(* POU GENERAL/ERROR/FB_InitErrorList, ST *)
FUNCTION_BLOCK FB_InitErrorList
VAR_INPUT
END_VAR
VAR_IN_OUT
	T_ErrorList:ST_ERROR_LIST;
END_VAR
VAR_OUTPUT
END_VAR
VAR
END_VAR
(* Static Deutsch Error List *)
T_ErrorList.asErrorListDeutsch.T_LanguagList[1]:='Fehler / Error während disable (Ausschalten) der Station';
T_ErrorList.asErrorListDeutsch.T_LanguagList[2]:='Nicht behandelter undefinierter Station Fehler';
T_ErrorList.asErrorListDeutsch.T_LanguagList[3]:='Z Achse-->Negativer HW Endschalter Aktiv';
T_ErrorList.asErrorListDeutsch.T_LanguagList[4]:='Z Achse-->Positiver HW Endschalter Aktiv';
T_ErrorList.asErrorListDeutsch.T_LanguagList[5]:='Z Achse-->Positiver + Negativer HW Endschalter Aktiv';
T_ErrorList.asErrorListDeutsch.T_LanguagList[6]:='AX5000 Parameter konnte nicht erfolgreich geschrieben werden';
T_ErrorList.asErrorListDeutsch.T_LanguagList[7]:='Achsen MasterModul2 konnte den Spindelkopf L Kanal 1 nicht finden';
T_ErrorList.asErrorListDeutsch.T_LanguagList[8]:='Kalibrierung-->ZylWzAuslenkung Sensor fehlerhaft';
T_ErrorList.asErrorListDeutsch.T_LanguagList[9]:='Z Achse muss referenziert sein';
T_ErrorList.asErrorListDeutsch.T_LanguagList[10]:='Achsen MasterModul2 konnte den Spindelkopf M Kanal 2 nicht finden';
T_ErrorList.asErrorListDeutsch.T_LanguagList[11]:='Hubprozesslänge > Z Mech EndPos';
T_ErrorList.asErrorListDeutsch.T_LanguagList[12]:='Ausfunkhub > Z Mech EndPos';
T_ErrorList.asErrorListDeutsch.T_LanguagList[13]:='Werkzeug ist nicht im Werkstück eingefädelt';
T_ErrorList.asErrorListDeutsch.T_LanguagList[14]:='Kühlmitteldruck ständig vorhanden';
T_ErrorList.asErrorListDeutsch.T_LanguagList[15]:='Fehler 15';
T_ErrorList.asErrorListDeutsch.T_LanguagList[16]:='Beim starten der Bearbeitung darf AuslenkSensor nicht ON sein';
T_ErrorList.asErrorListDeutsch.T_LanguagList[17]:='Beim starten der Bearbeitung darf DrehmSensorHC nicht ON sein';
T_ErrorList.asErrorListDeutsch.T_LanguagList[18]:='Z LadePos > Z Mech EndPos';
T_ErrorList.asErrorListDeutsch.T_LanguagList[19]:='Z Bearb StartPos > Z Mech EndPos';
T_ErrorList.asErrorListDeutsch.T_LanguagList[20]:='Z Bearb EndPos > Z Mech EndPos';
T_ErrorList.asErrorListDeutsch.T_LanguagList[21]:='Z WzWechsel Pos > Z Mech EndPos';
T_ErrorList.asErrorListDeutsch.T_LanguagList[22]:='Z LadePos: Stimmt nicht mit anderen Positionen überein';
T_ErrorList.asErrorListDeutsch.T_LanguagList[23]:='Z Bearb StartPos: Stimmt nicht mit anderen Positionen überein';
T_ErrorList.asErrorListDeutsch.T_LanguagList[24]:='Z Bearb EndPos: Stimmt nicht mit anderen Positionen überein';
T_ErrorList.asErrorListDeutsch.T_LanguagList[25]:='Kalibrierung-->ZylWzAuslenkung Zylinder blockiert';
T_ErrorList.asErrorListDeutsch.T_LanguagList[26]:='Kalibrierung-->ZylWzAuslenkung Sensor fehlerhaft';
T_ErrorList.asErrorListDeutsch.T_LanguagList[27]:='Fehler 27';
T_ErrorList.asErrorListDeutsch.T_LanguagList[28]:='Wz Drehmoment Max überschritten';
T_ErrorList.asErrorListDeutsch.T_LanguagList[29]:='Wz Drehmoment Überlast Aktiv';
T_ErrorList.asErrorListDeutsch.T_LanguagList[30]:='Beim Zentrieren muss der ZylWstkEntspannen auf BearbeitPos sein';
T_ErrorList.asErrorListDeutsch.T_LanguagList[31]:='Z Bearb EndPos Berechn. > Z Bearb EndPos Max';
T_ErrorList.asErrorListDeutsch.T_LanguagList[32]:='Z ZentrierPos berechn. > Z Mech EndPos';
T_ErrorList.asErrorListDeutsch.T_LanguagList[33]:='Zentrier EndPos > Z Mech EndPos';
T_ErrorList.asErrorListDeutsch.T_LanguagList[34]:='Z ZentrierPos berechn. > Z Bearb EndPos Max';
T_ErrorList.asErrorListDeutsch.T_LanguagList[35]:='Z WzZylinder Pos > Z Mech EndPos';
T_ErrorList.asErrorListDeutsch.T_LanguagList[36]:='Beim zylindrischer Teil wurde die Max EndPos erreicht';
T_ErrorList.asErrorListDeutsch.T_LanguagList[37]:='Fehler 37';
T_ErrorList.asErrorListDeutsch.T_LanguagList[38]:='Fehler 38';
T_ErrorList.asErrorListDeutsch.T_LanguagList[39]:='Fehler 39';
T_ErrorList.asErrorListDeutsch.T_LanguagList[40]:='Fehler 40';
T_ErrorList.asErrorListDeutsch.T_LanguagList[41]:='Fehler 41';
T_ErrorList.asErrorListDeutsch.T_LanguagList[42]:='Fehler 42';
T_ErrorList.asErrorListDeutsch.T_LanguagList[43]:='Fehler 43';
T_ErrorList.asErrorListDeutsch.T_LanguagList[44]:='Fehler 44';
T_ErrorList.asErrorListDeutsch.T_LanguagList[45]:='Fehler 45';
T_ErrorList.asErrorListDeutsch.T_LanguagList[46]:='Fehler 46';
T_ErrorList.asErrorListDeutsch.T_LanguagList[47]:='Fehler 47';
T_ErrorList.asErrorListDeutsch.T_LanguagList[48]:='WzWechsel muss vorgenommen werden';
T_ErrorList.asErrorListDeutsch.T_LanguagList[49]:='Datei für zu ladendes Profil nicht gefunden';
T_ErrorList.asErrorListDeutsch.T_LanguagList[50]:='Fehler 50';
T_ErrorList.asErrorListDeutsch.T_LanguagList[51]:='Profilname von Datei ist anders als geladenes Profil';
T_ErrorList.asErrorListDeutsch.T_LanguagList[52]:='Syntaxfehler von zu ladendes Profil';
T_ErrorList.asErrorListDeutsch.T_LanguagList[53]:='Fehler 53';
T_ErrorList.asErrorListDeutsch.T_LanguagList[54]:='Profil konnte nicht gespeichert werden da Verzeichnis fehlt';
T_ErrorList.asErrorListDeutsch.T_LanguagList[55]:='Kalibrierung-->ZylWzDrehmHC Sensor fehlerhaft';
T_ErrorList.asErrorListDeutsch.T_LanguagList[56]:='Kalibrierung-->ZylWzAuslenkung+ZylWzDrehmHC Sensor fehlerhaft';
T_ErrorList.asErrorListDeutsch.T_LanguagList[57]:='Kalibrierung-->ZylWzDrehmHC Zylinder blockiert';
T_ErrorList.asErrorListDeutsch.T_LanguagList[58]:='Kalibrierung-->ZylWzAuslenkung+ZylWzDrehmHC Zylinder blockiert';
T_ErrorList.asErrorListDeutsch.T_LanguagList[59]:='Beim starten der Bearbeitung darf DrehmSensorHCÜberlast nicht ON sein';
T_ErrorList.asErrorListDeutsch.T_LanguagList[60]:='Zentrierproz. HC1 eingetroffen';
T_ErrorList.asErrorListDeutsch.T_LanguagList[61]:='Zentrierproz. StartPos erreicht und HC2 immer noch ON';
T_ErrorList.asErrorListDeutsch.T_LanguagList[62]:='Fehler 62';
T_ErrorList.asErrorListDeutsch.T_LanguagList[63]:='Fehler 63';
T_ErrorList.asErrorListDeutsch.T_LanguagList[64]:='Fehler 64';
T_ErrorList.asErrorListDeutsch.T_LanguagList[65]:='Fehler 65';
T_ErrorList.asErrorListDeutsch.T_LanguagList[66]:='Aufgerufene Achsfunktion besteht nicht';
T_ErrorList.asErrorListDeutsch.T_LanguagList[67]:='Achsfunktion nicht ausführbar wenn Stop-Funktion Aktiv';
T_ErrorList.asErrorListDeutsch.T_LanguagList[68]:='Fehler 68';
T_ErrorList.asErrorListDeutsch.T_LanguagList[69]:='Fehler 69';
T_ErrorList.asErrorListDeutsch.T_LanguagList[70]:='Fehler 70';
T_ErrorList.asErrorListDeutsch.T_LanguagList[71]:='Fehler 71';
T_ErrorList.asErrorListDeutsch.T_LanguagList[72]:='Fehler 72';
T_ErrorList.asErrorListDeutsch.T_LanguagList[73]:='Fehler 73';
T_ErrorList.asErrorListDeutsch.T_LanguagList[74]:='Fehler 74';
T_ErrorList.asErrorListDeutsch.T_LanguagList[75]:='(Schleppabstandsüberschreitung)';
T_ErrorList.asErrorListDeutsch.T_LanguagList[76]:='Not Aus Taste Maschine wurde gedrückt';
T_ErrorList.asErrorListDeutsch.T_LanguagList[77]:='Fehler 77';
T_ErrorList.asErrorListDeutsch.T_LanguagList[78]:='Fehler 78';
T_ErrorList.asErrorListDeutsch.T_LanguagList[79]:='Fehler 79';
T_ErrorList.asErrorListDeutsch.T_LanguagList[80]:='Fehler 80';
T_ErrorList.asErrorListDeutsch.T_LanguagList[81]:='Fehler 81';
T_ErrorList.asErrorListDeutsch.T_LanguagList[82]:='Fehler 82';
T_ErrorList.asErrorListDeutsch.T_LanguagList[83]:='Keine Druckluft';
T_ErrorList.asErrorListDeutsch.T_LanguagList[84]:='EtherCAT 1 Klemme Fehlerhaft';
T_ErrorList.asErrorListDeutsch.T_LanguagList[85]:='EtherCAT 2 Klemme Fehlerhaft';
T_ErrorList.asErrorListDeutsch.T_LanguagList[86]:='Maxon EPOS nicht im Operational Mode OP';
T_ErrorList.asErrorListDeutsch.T_LanguagList[87]:='SMC Ventilinsel nicht im Operational Mode OP';
T_ErrorList.asErrorListDeutsch.T_LanguagList[88]:='Achsen MasterModul 1 nicht im Operational Mode OP';
T_ErrorList.asErrorListDeutsch.T_LanguagList[89]:='Achsen MasterModul 2 nicht im Operational Mode OP';
T_ErrorList.asErrorListDeutsch.T_LanguagList[90]:='Spannungsversorgung 24VDC fehlerhaft';
T_ErrorList.asErrorListDeutsch.T_LanguagList[91]:='Fehler 91';
T_ErrorList.asErrorListDeutsch.T_LanguagList[92]:='Fehler 92';
T_ErrorList.asErrorListDeutsch.T_LanguagList[93]:='Fehler 93';
T_ErrorList.asErrorListDeutsch.T_LanguagList[94]:='Fehler 94';
T_ErrorList.asErrorListDeutsch.T_LanguagList[95]:='Fehler 95';
T_ErrorList.asErrorListDeutsch.T_LanguagList[96]:='Fehler 96';
T_ErrorList.asErrorListDeutsch.T_LanguagList[97]:='Fehler 97';
T_ErrorList.asErrorListDeutsch.T_LanguagList[98]:='USB-Stick konnte nicht gefunden werden für Profil lesen/schreiben';
T_ErrorList.asErrorListDeutsch.T_LanguagList[99]:='USB-Stick konnte nicht gefunden werden für Profil löschen';
T_ErrorList.asErrorListDeutsch.T_LanguagList[100]:='Spannungsversorgung wurde ausgeschaltet';
T_ErrorList.asErrorListDeutsch.T_LanguagList[101]:='Syntaxfehler mindestens einer Profildatei beim lesen aller Profile';
T_ErrorList.asErrorListDeutsch.T_LanguagList[102]:='NovRAM Speicher Fehlerhaft';
T_ErrorList.asErrorListDeutsch.T_LanguagList[103]:='Nicht behandelter undefinierter Prozess Fehler';
T_ErrorList.asErrorListDeutsch.T_LanguagList[104]:='USB-Stick konnte nicht gefunden werden';
T_ErrorList.asErrorListDeutsch.T_LanguagList[105]:='Zylinder Funktion nicht implementiert';
T_ErrorList.asErrorListDeutsch.T_LanguagList[106]:='Zylinder Aktiv-->Sensor nicht ON';
T_ErrorList.asErrorListDeutsch.T_LanguagList[107]:='Zylinder Inaktiv-->Sensor nicht ON';
T_ErrorList.asErrorListDeutsch.T_LanguagList[108]:='Nicht behandelter undefinierter Zylinder Fehler';
T_ErrorList.asErrorListDeutsch.T_LanguagList[109]:='Bremse Aktiv von ST1';
T_ErrorList.asErrorListDeutsch.T_LanguagList[110]:='Fehler 110';
T_ErrorList.asErrorListDeutsch.T_LanguagList[111]:='Fehler 111';
T_ErrorList.asErrorListDeutsch.T_LanguagList[112]:='Fehler 112';
T_ErrorList.asErrorListDeutsch.T_LanguagList[113]:='Fehler 113';
T_ErrorList.asErrorListDeutsch.T_LanguagList[114]:='Fehler 114';
T_ErrorList.asErrorListDeutsch.T_LanguagList[115]:='Fehler 115';
T_ErrorList.asErrorListDeutsch.T_LanguagList[116]:='Fehler 116';
T_ErrorList.asErrorListDeutsch.T_LanguagList[117]:='Fehler 117';
T_ErrorList.asErrorListDeutsch.T_LanguagList[118]:='Fehler 118';
T_ErrorList.asErrorListDeutsch.T_LanguagList[119]:='Fehler 119';
T_ErrorList.asErrorListDeutsch.T_LanguagList[120]:='Fehler 120';
T_ErrorList.asErrorListDeutsch.T_LanguagList[121]:='Fehler 121';
T_ErrorList.asErrorListDeutsch.T_LanguagList[122]:='Fehler 122';
T_ErrorList.asErrorListDeutsch.T_LanguagList[123]:='Fehler 123';
T_ErrorList.asErrorListDeutsch.T_LanguagList[124]:='Fehler 124';
T_ErrorList.asErrorListDeutsch.T_LanguagList[125]:='Fehler 125';
T_ErrorList.asErrorListDeutsch.T_LanguagList[126]:='Fehler 126';
T_ErrorList.asErrorListDeutsch.T_LanguagList[127]:='Fehler 127';
T_ErrorList.asErrorListDeutsch.T_LanguagList[128]:='Fehler 128';
T_ErrorList.asErrorListDeutsch.T_LanguagList[129]:='Fehler 129';
T_ErrorList.asErrorListDeutsch.T_LanguagList[130]:='Fehler 130';
T_ErrorList.asErrorListDeutsch.T_LanguagList[131]:='Fehler 131';
T_ErrorList.asErrorListDeutsch.T_LanguagList[132]:='Fehler 132';
T_ErrorList.asErrorListDeutsch.T_LanguagList[133]:='Fehler 133';
T_ErrorList.asErrorListDeutsch.T_LanguagList[134]:='Fehler 134';
T_ErrorList.asErrorListDeutsch.T_LanguagList[135]:='Fehler 135';
T_ErrorList.asErrorListDeutsch.T_LanguagList[136]:='Fehler 136';
T_ErrorList.asErrorListDeutsch.T_LanguagList[137]:='Fehler 137';
T_ErrorList.asErrorListDeutsch.T_LanguagList[138]:='Fehler 138';
T_ErrorList.asErrorListDeutsch.T_LanguagList[139]:='Fehler 139';
T_ErrorList.asErrorListDeutsch.T_LanguagList[140]:='Fehler 140';
T_ErrorList.asErrorListDeutsch.T_LanguagList[141]:='Fehler 141';
T_ErrorList.asErrorListDeutsch.T_LanguagList[142]:='Fehler 142';
T_ErrorList.asErrorListDeutsch.T_LanguagList[143]:='Fehler 143';
T_ErrorList.asErrorListDeutsch.T_LanguagList[144]:='Fehler 144';
T_ErrorList.asErrorListDeutsch.T_LanguagList[145]:='Fehler 145';
T_ErrorList.asErrorListDeutsch.T_LanguagList[146]:='HDD steht nicht Bereit';
T_ErrorList.asErrorListDeutsch.T_LanguagList[147]:='Timeout beim Schreiben auf USB-Stick';
T_ErrorList.asErrorListDeutsch.T_LanguagList[148]:='USB Stick nicht schreibbar';
T_ErrorList.asErrorListDeutsch.T_LanguagList[149]:='USB Stick nicht gefunden';
T_ErrorList.asErrorListDeutsch.T_LanguagList[150]:='Fehler 150';
T_ErrorList.asErrorListDeutsch.T_LanguagList[151]:='Fehler 151';
T_ErrorList.asErrorListDeutsch.T_LanguagList[152]:='Fehler 152';
T_ErrorList.asErrorListDeutsch.T_LanguagList[153]:='Fehler 153';
T_ErrorList.asErrorListDeutsch.T_LanguagList[154]:='Fehler 154';
T_ErrorList.asErrorListDeutsch.T_LanguagList[155]:='Fehler 155';
T_ErrorList.asErrorListDeutsch.T_LanguagList[156]:='Fehler 156';
T_ErrorList.asErrorListDeutsch.T_LanguagList[157]:='Fehler 157';
T_ErrorList.asErrorListDeutsch.T_LanguagList[158]:='Fehler 158';
T_ErrorList.asErrorListDeutsch.T_LanguagList[159]:='Fehler 159';
T_ErrorList.asErrorListDeutsch.T_LanguagList[160]:='Fehler 160';
T_ErrorList.asErrorListDeutsch.T_LanguagList[161]:='Fehler 161';
T_ErrorList.asErrorListDeutsch.T_LanguagList[162]:='Fehler 162';
T_ErrorList.asErrorListDeutsch.T_LanguagList[163]:='Fehler 163';
T_ErrorList.asErrorListDeutsch.T_LanguagList[164]:='Fehler 164';
T_ErrorList.asErrorListDeutsch.T_LanguagList[165]:='Fehler 165';
T_ErrorList.asErrorListDeutsch.T_LanguagList[166]:='Fehler 166';
T_ErrorList.asErrorListDeutsch.T_LanguagList[167]:='Fehler 167';
T_ErrorList.asErrorListDeutsch.T_LanguagList[168]:='Fehler 168';
T_ErrorList.asErrorListDeutsch.T_LanguagList[169]:='Fehler 169';
T_ErrorList.asErrorListDeutsch.T_LanguagList[170]:='Fehler 170';
T_ErrorList.asErrorListDeutsch.T_LanguagList[171]:='Fehler 171';
T_ErrorList.asErrorListDeutsch.T_LanguagList[172]:='Fehler 172';
T_ErrorList.asErrorListDeutsch.T_LanguagList[173]:='Fehler 173';
T_ErrorList.asErrorListDeutsch.T_LanguagList[174]:='Fehler 174';
T_ErrorList.asErrorListDeutsch.T_LanguagList[175]:='Fehler 175';
T_ErrorList.asErrorListDeutsch.T_LanguagList[176]:='Fehler 176';
T_ErrorList.asErrorListDeutsch.T_LanguagList[177]:='Fehler 177';
T_ErrorList.asErrorListDeutsch.T_LanguagList[178]:='Fehler 178';
T_ErrorList.asErrorListDeutsch.T_LanguagList[179]:='Fehler 179';
T_ErrorList.asErrorListDeutsch.T_LanguagList[180]:='Fehler 180';
T_ErrorList.asErrorListDeutsch.T_LanguagList[181]:='Fehler 181';
T_ErrorList.asErrorListDeutsch.T_LanguagList[182]:='Fehler 182';
T_ErrorList.asErrorListDeutsch.T_LanguagList[183]:='Fehler 183';
T_ErrorList.asErrorListDeutsch.T_LanguagList[184]:='Fehler 184';
T_ErrorList.asErrorListDeutsch.T_LanguagList[185]:='Fehler 185';
T_ErrorList.asErrorListDeutsch.T_LanguagList[186]:='Fehler 186';
T_ErrorList.asErrorListDeutsch.T_LanguagList[187]:='Fehler 187';
T_ErrorList.asErrorListDeutsch.T_LanguagList[188]:='Fehler 188';
T_ErrorList.asErrorListDeutsch.T_LanguagList[189]:='Fehler 189';
T_ErrorList.asErrorListDeutsch.T_LanguagList[190]:='Fehler 190';
T_ErrorList.asErrorListDeutsch.T_LanguagList[191]:='Fehler 191';
T_ErrorList.asErrorListDeutsch.T_LanguagList[192]:='Fehler 192';
T_ErrorList.asErrorListDeutsch.T_LanguagList[193]:='Fehler 193';
T_ErrorList.asErrorListDeutsch.T_LanguagList[194]:='Fehler 194';
T_ErrorList.asErrorListDeutsch.T_LanguagList[195]:='Fehler 195';
T_ErrorList.asErrorListDeutsch.T_LanguagList[196]:='Fehler 196';
T_ErrorList.asErrorListDeutsch.T_LanguagList[197]:='Fehler 197';
T_ErrorList.asErrorListDeutsch.T_LanguagList[198]:='Fehler 198';
T_ErrorList.asErrorListDeutsch.T_LanguagList[199]:='Fehler 199';
T_ErrorList.asErrorListDeutsch.T_LanguagList[200]:='Fehler 200';
T_ErrorList.asErrorListDeutsch.T_LanguagList[201]:='Fehler 201';
T_ErrorList.asErrorListDeutsch.T_LanguagList[202]:='Fehler 202';
T_ErrorList.asErrorListDeutsch.T_LanguagList[203]:='Fehler 203';
T_ErrorList.asErrorListDeutsch.T_LanguagList[204]:='Fehler 204';
T_ErrorList.asErrorListDeutsch.T_LanguagList[205]:='Fehler 205';
T_ErrorList.asErrorListDeutsch.T_LanguagList[206]:='Fehler 206';
T_ErrorList.asErrorListDeutsch.T_LanguagList[207]:='Fehler 207';
T_ErrorList.asErrorListDeutsch.T_LanguagList[208]:='Fehler 208';
T_ErrorList.asErrorListDeutsch.T_LanguagList[209]:='Fehler 209';
T_ErrorList.asErrorListDeutsch.T_LanguagList[210]:='Fehler 210';
T_ErrorList.asErrorListDeutsch.T_LanguagList[211]:='Fehler 211';
T_ErrorList.asErrorListDeutsch.T_LanguagList[212]:='Fehler 212';
T_ErrorList.asErrorListDeutsch.T_LanguagList[213]:='Fehler 213';
T_ErrorList.asErrorListDeutsch.T_LanguagList[214]:='Fehler 214';
T_ErrorList.asErrorListDeutsch.T_LanguagList[215]:='Fehler 215';
T_ErrorList.asErrorListDeutsch.T_LanguagList[216]:='Fehler 216';
T_ErrorList.asErrorListDeutsch.T_LanguagList[217]:='Fehler 217';
T_ErrorList.asErrorListDeutsch.T_LanguagList[218]:='Fehler 218';
T_ErrorList.asErrorListDeutsch.T_LanguagList[219]:='Fehler 219';
T_ErrorList.asErrorListDeutsch.T_LanguagList[220]:='Fehler 220';
T_ErrorList.asErrorListDeutsch.T_LanguagList[221]:='Fehler 221';
T_ErrorList.asErrorListDeutsch.T_LanguagList[222]:='Fehler 222';
T_ErrorList.asErrorListDeutsch.T_LanguagList[223]:='Fehler 223';
T_ErrorList.asErrorListDeutsch.T_LanguagList[224]:='Fehler 224';
T_ErrorList.asErrorListDeutsch.T_LanguagList[225]:='Fehler 225';
T_ErrorList.asErrorListDeutsch.T_LanguagList[226]:='Fehler 226';
T_ErrorList.asErrorListDeutsch.T_LanguagList[227]:='Fehler 227';
T_ErrorList.asErrorListDeutsch.T_LanguagList[228]:='Fehler 228';
T_ErrorList.asErrorListDeutsch.T_LanguagList[229]:='Fehler 229';
T_ErrorList.asErrorListDeutsch.T_LanguagList[230]:='Fehler 230';
T_ErrorList.asErrorListDeutsch.T_LanguagList[231]:='Fehler 231';
T_ErrorList.asErrorListDeutsch.T_LanguagList[232]:='Fehler 232';
T_ErrorList.asErrorListDeutsch.T_LanguagList[233]:='Fehler 233';
T_ErrorList.asErrorListDeutsch.T_LanguagList[234]:='Fehler 234';
T_ErrorList.asErrorListDeutsch.T_LanguagList[235]:='Fehler 235';
T_ErrorList.asErrorListDeutsch.T_LanguagList[236]:='Fehler 236';
T_ErrorList.asErrorListDeutsch.T_LanguagList[237]:='Fehler 237';
T_ErrorList.asErrorListDeutsch.T_LanguagList[238]:='Fehler 238';
T_ErrorList.asErrorListDeutsch.T_LanguagList[239]:='Fehler 239';
T_ErrorList.asErrorListDeutsch.T_LanguagList[240]:='Fehler 240';
T_ErrorList.asErrorListDeutsch.T_LanguagList[241]:='Fehler 241';
T_ErrorList.asErrorListDeutsch.T_LanguagList[242]:='Fehler 242';
T_ErrorList.asErrorListDeutsch.T_LanguagList[243]:='Fehler 243';
T_ErrorList.asErrorListDeutsch.T_LanguagList[244]:='Fehler 244';
T_ErrorList.asErrorListDeutsch.T_LanguagList[245]:='Fehler 245';
T_ErrorList.asErrorListDeutsch.T_LanguagList[246]:='Fehler 246';
T_ErrorList.asErrorListDeutsch.T_LanguagList[247]:='Fehler 247';
T_ErrorList.asErrorListDeutsch.T_LanguagList[248]:='Fehler 248';
T_ErrorList.asErrorListDeutsch.T_LanguagList[249]:='Fehler 249';
T_ErrorList.asErrorListDeutsch.T_LanguagList[250]:='Fehler 250';
T_ErrorList.asErrorListDeutsch.T_LanguagList[251]:='Fehler 251';
T_ErrorList.asErrorListDeutsch.T_LanguagList[252]:='Fehler 252';
T_ErrorList.asErrorListDeutsch.T_LanguagList[253]:='Fehler 253';
T_ErrorList.asErrorListDeutsch.T_LanguagList[254]:='Fehler 254';
T_ErrorList.asErrorListDeutsch.T_LanguagList[255]:='Fehler 255';
T_ErrorList.asErrorListDeutsch.T_LanguagList[256]:='Fehler 256';
T_ErrorList.asErrorListDeutsch.T_LanguagList[257]:='Fehler 257';
T_ErrorList.asErrorListDeutsch.T_LanguagList[258]:='Fehler 258';
T_ErrorList.asErrorListDeutsch.T_LanguagList[259]:='Fehler 259';
T_ErrorList.asErrorListDeutsch.T_LanguagList[260]:='Fehler 260';
T_ErrorList.asErrorListDeutsch.T_LanguagList[261]:='Fehler 261';
T_ErrorList.asErrorListDeutsch.T_LanguagList[262]:='Fehler 262';
T_ErrorList.asErrorListDeutsch.T_LanguagList[263]:='Fehler 263';
T_ErrorList.asErrorListDeutsch.T_LanguagList[264]:='Fehler 264';
T_ErrorList.asErrorListDeutsch.T_LanguagList[265]:='Fehler 265';
T_ErrorList.asErrorListDeutsch.T_LanguagList[266]:='Fehler 266';
T_ErrorList.asErrorListDeutsch.T_LanguagList[267]:='Fehler 267';
T_ErrorList.asErrorListDeutsch.T_LanguagList[268]:='Fehler 268';
T_ErrorList.asErrorListDeutsch.T_LanguagList[269]:='Fehler 269';
T_ErrorList.asErrorListDeutsch.T_LanguagList[270]:='Fehler 270';
T_ErrorList.asErrorListDeutsch.T_LanguagList[271]:='Fehler 271';
T_ErrorList.asErrorListDeutsch.T_LanguagList[272]:='Fehler 272';
T_ErrorList.asErrorListDeutsch.T_LanguagList[273]:='Fehler 273';
T_ErrorList.asErrorListDeutsch.T_LanguagList[274]:='Fehler 274';
T_ErrorList.asErrorListDeutsch.T_LanguagList[275]:='Fehler 275';
T_ErrorList.asErrorListDeutsch.T_LanguagList[276]:='Fehler 276';
T_ErrorList.asErrorListDeutsch.T_LanguagList[277]:='Fehler 277';
T_ErrorList.asErrorListDeutsch.T_LanguagList[278]:='Fehler 278';
T_ErrorList.asErrorListDeutsch.T_LanguagList[279]:='Fehler 279';
T_ErrorList.asErrorListDeutsch.T_LanguagList[280]:='Fehler 280';
T_ErrorList.asErrorListDeutsch.T_LanguagList[281]:='Fehler 281';
T_ErrorList.asErrorListDeutsch.T_LanguagList[282]:='Fehler 282';
T_ErrorList.asErrorListDeutsch.T_LanguagList[283]:='Fehler 283';
T_ErrorList.asErrorListDeutsch.T_LanguagList[284]:='Fehler 284';
T_ErrorList.asErrorListDeutsch.T_LanguagList[285]:='Fehler 285';
T_ErrorList.asErrorListDeutsch.T_LanguagList[286]:='Fehler 286';
T_ErrorList.asErrorListDeutsch.T_LanguagList[287]:='Fehler 287';
T_ErrorList.asErrorListDeutsch.T_LanguagList[288]:='Fehler 288';
T_ErrorList.asErrorListDeutsch.T_LanguagList[289]:='Fehler 289';
T_ErrorList.asErrorListDeutsch.T_LanguagList[290]:='Fehler 290';
T_ErrorList.asErrorListDeutsch.T_LanguagList[291]:='Fehler 291';
T_ErrorList.asErrorListDeutsch.T_LanguagList[292]:='Fehler 292';
T_ErrorList.asErrorListDeutsch.T_LanguagList[293]:='Fehler 293';
T_ErrorList.asErrorListDeutsch.T_LanguagList[294]:='Fehler 294';
T_ErrorList.asErrorListDeutsch.T_LanguagList[295]:='Fehler 295';
T_ErrorList.asErrorListDeutsch.T_LanguagList[296]:='Fehler 296';
T_ErrorList.asErrorListDeutsch.T_LanguagList[297]:='Fehler 297';
T_ErrorList.asErrorListDeutsch.T_LanguagList[298]:='Fehler 298';
T_ErrorList.asErrorListDeutsch.T_LanguagList[299]:='Fehler 299';
T_ErrorList.asErrorListDeutsch.T_LanguagList[300]:='Fehler 300';

(* Static English Error List *)
T_ErrorList.asErrorListEnglish.T_LanguagList[1]:='Error while disable of the Station';
T_ErrorList.asErrorListEnglish.T_LanguagList[2]:='Not handled undefined Station Error';
T_ErrorList.asErrorListEnglish.T_LanguagList[3]:='Z Axis-->Negative HW limit switch Active';
T_ErrorList.asErrorListEnglish.T_LanguagList[4]:='Z Axis-->Positive HW limit switch Active';
T_ErrorList.asErrorListEnglish.T_LanguagList[5]:='Z Axis-->Positive + Negative HW limit switch Active';
T_ErrorList.asErrorListEnglish.T_LanguagList[6]:='AX5000 Parameter could not be written successfully';
T_ErrorList.asErrorListEnglish.T_LanguagList[7]:='Axis MasterModul2 could not find spindle head L channel 1';
T_ErrorList.asErrorListEnglish.T_LanguagList[8]:='Calibration-->CylToolDeflection Sensor failure';
T_ErrorList.asErrorListEnglish.T_LanguagList[9]:='Z Axis must be referenced';
T_ErrorList.asErrorListEnglish.T_LanguagList[10]:='Axis MasterModul2 could not find spindle head M channel 2';
T_ErrorList.asErrorListEnglish.T_LanguagList[11]:='Z Process stroke > Z Mech EndPos';
T_ErrorList.asErrorListEnglish.T_LanguagList[12]:='Spark-out > Z Mech EndPos';
T_ErrorList.asErrorListEnglish.T_LanguagList[13]:='Tool is not Infeeded into the Workpiece';
T_ErrorList.asErrorListEnglish.T_LanguagList[14]:='Coolant pressure still ON';
T_ErrorList.asErrorListEnglish.T_LanguagList[15]:='Error 15';
T_ErrorList.asErrorListEnglish.T_LanguagList[16]:='During starting of the Working could not be ON the ToolDeflection Sensor';
T_ErrorList.asErrorListEnglish.T_LanguagList[17]:='During starting of the Working could not be ON the ToolTorque Sensor';
T_ErrorList.asErrorListEnglish.T_LanguagList[18]:='Z LoadPos > Z Mech EndPos';
T_ErrorList.asErrorListEnglish.T_LanguagList[19]:='Z Work StartPos > Z Mech EndPos';
T_ErrorList.asErrorListEnglish.T_LanguagList[20]:='Z Work EndPos > Z Mech EndPos';
T_ErrorList.asErrorListEnglish.T_LanguagList[21]:='Z ToolChange Pos > Z Mech EndPos';
T_ErrorList.asErrorListEnglish.T_LanguagList[22]:='Z LoadPos: Discrepancy with other Z Position';
T_ErrorList.asErrorListEnglish.T_LanguagList[23]:='Z Work StartPos: Discrepancy with other Z Position';
T_ErrorList.asErrorListEnglish.T_LanguagList[24]:='Z Work EndPos: Discrepancy with other Z Position';
T_ErrorList.asErrorListEnglish.T_LanguagList[25]:='Calibration-->CylToolDeflection Cylinder is blocked';
T_ErrorList.asErrorListEnglish.T_LanguagList[26]:='Calibration-->CylToolDeflection Sensor failure';
T_ErrorList.asErrorListEnglish.T_LanguagList[27]:='Error 27';
T_ErrorList.asErrorListEnglish.T_LanguagList[28]:='ToolTorque Max exceed';
T_ErrorList.asErrorListEnglish.T_LanguagList[29]:='ToolTorque Overload Active';
T_ErrorList.asErrorListEnglish.T_LanguagList[30]:='When centring, the CylWPUnfix must be to WorkPosition';
T_ErrorList.asErrorListEnglish.T_LanguagList[31]:='Z Work EndPos calc. > Z Work EndPos Max';
T_ErrorList.asErrorListEnglish.T_LanguagList[32]:='Z Centring Pos calc. > Z Mech EndPos';
T_ErrorList.asErrorListEnglish.T_LanguagList[33]:='Z Centring EndPos > Z Mech EndPos';
T_ErrorList.asErrorListEnglish.T_LanguagList[34]:='Z Centring Pos calc. > Z Work EndPos Max';
T_ErrorList.asErrorListEnglish.T_LanguagList[35]:='Z ToolCylindrical Pos > Z Mech EndPos';
T_ErrorList.asErrorListEnglish.T_LanguagList[36]:='On cylindrical part was reach the max EndPos';
T_ErrorList.asErrorListEnglish.T_LanguagList[37]:='Error 37';
T_ErrorList.asErrorListEnglish.T_LanguagList[38]:='Error 38';
T_ErrorList.asErrorListEnglish.T_LanguagList[39]:='Error 39';
T_ErrorList.asErrorListEnglish.T_LanguagList[40]:='Error 40';
T_ErrorList.asErrorListEnglish.T_LanguagList[41]:='Error 41';
T_ErrorList.asErrorListEnglish.T_LanguagList[42]:='Error 42';
T_ErrorList.asErrorListEnglish.T_LanguagList[43]:='Error 43';
T_ErrorList.asErrorListEnglish.T_LanguagList[44]:='Error 44';
T_ErrorList.asErrorListEnglish.T_LanguagList[45]:='Error 45';
T_ErrorList.asErrorListEnglish.T_LanguagList[46]:='Error 46';
T_ErrorList.asErrorListEnglish.T_LanguagList[47]:='Error 47';
T_ErrorList.asErrorListEnglish.T_LanguagList[48]:='Tool must be changed';
T_ErrorList.asErrorListEnglish.T_LanguagList[49]:='File for to load Profile not found';
T_ErrorList.asErrorListEnglish.T_LanguagList[50]:='Error 50';
T_ErrorList.asErrorListEnglish.T_LanguagList[51]:='Profile name of File is different as loaded Profile';
T_ErrorList.asErrorListEnglish.T_LanguagList[52]:='Syntax Error of to load Profile';
T_ErrorList.asErrorListEnglish.T_LanguagList[53]:='Error 53';
T_ErrorList.asErrorListEnglish.T_LanguagList[54]:='Profile not saved because the directory is missing';
T_ErrorList.asErrorListEnglish.T_LanguagList[55]:='Calibration-->CylToolTorque Sensor failure';
T_ErrorList.asErrorListEnglish.T_LanguagList[56]:='Calibration-->CylToolDeflection+CylToolTorque Sensor failure';
T_ErrorList.asErrorListEnglish.T_LanguagList[57]:='Calibration-->CylToolTorque Cylinder is blocked';
T_ErrorList.asErrorListEnglish.T_LanguagList[58]:='Calibration-->CylToolDeflection+CylToolTorque Cylinder is blocked';
T_ErrorList.asErrorListEnglish.T_LanguagList[59]:='During starting of the Working could not be ON the ToolTorque Overload Sensor';
T_ErrorList.asErrorListEnglish.T_LanguagList[60]:='Centring Process HC1 active';
T_ErrorList.asErrorListEnglish.T_LanguagList[61]:='Centring Proc. StartPos reach and HC2 still ON';
T_ErrorList.asErrorListEnglish.T_LanguagList[62]:='Error 62';
T_ErrorList.asErrorListEnglish.T_LanguagList[63]:='Error 63';
T_ErrorList.asErrorListEnglish.T_LanguagList[64]:='Error 64';
T_ErrorList.asErrorListEnglish.T_LanguagList[65]:='Error 65';
T_ErrorList.asErrorListEnglish.T_LanguagList[66]:='Called Axis function do not exist';
T_ErrorList.asErrorListEnglish.T_LanguagList[67]:='Axis function not executable during Stopp- function is Active';
T_ErrorList.asErrorListEnglish.T_LanguagList[68]:='Error 68';
T_ErrorList.asErrorListEnglish.T_LanguagList[69]:='Error 69';
T_ErrorList.asErrorListEnglish.T_LanguagList[70]:='Error 70';
T_ErrorList.asErrorListEnglish.T_LanguagList[71]:='Error 71';
T_ErrorList.asErrorListEnglish.T_LanguagList[72]:='Error 72';
T_ErrorList.asErrorListEnglish.T_LanguagList[73]:='Error 73';
T_ErrorList.asErrorListEnglish.T_LanguagList[74]:='Error 74';
T_ErrorList.asErrorListEnglish.T_LanguagList[75]:='(Position drag excess)';
T_ErrorList.asErrorListEnglish.T_LanguagList[76]:='Emergency Button Machine pressed';
T_ErrorList.asErrorListEnglish.T_LanguagList[77]:='Error 77';
T_ErrorList.asErrorListEnglish.T_LanguagList[78]:='Error 78';
T_ErrorList.asErrorListEnglish.T_LanguagList[79]:='Error 79';
T_ErrorList.asErrorListEnglish.T_LanguagList[80]:='Error 80';
T_ErrorList.asErrorListEnglish.T_LanguagList[81]:='Error 81';
T_ErrorList.asErrorListEnglish.T_LanguagList[82]:='Error 82';
T_ErrorList.asErrorListEnglish.T_LanguagList[83]:='No air pressure';
T_ErrorList.asErrorListEnglish.T_LanguagList[84]:='EtherCAT 1 Terminal failure';
T_ErrorList.asErrorListEnglish.T_LanguagList[85]:='EtherCAT 2 Terminal failure';
T_ErrorList.asErrorListEnglish.T_LanguagList[86]:='Maxon EPOS not in Operational Mode OP';
T_ErrorList.asErrorListEnglish.T_LanguagList[87]:='SMC Valve not in Operational Mode OP';
T_ErrorList.asErrorListEnglish.T_LanguagList[88]:='Axis MasterModul 1 not in Operational Mode OP';
T_ErrorList.asErrorListEnglish.T_LanguagList[89]:='Axis MasterModul 2 not in Operational Mode OP';
T_ErrorList.asErrorListEnglish.T_LanguagList[90]:='Power 24VDC failure';
T_ErrorList.asErrorListEnglish.T_LanguagList[91]:='Error 91';
T_ErrorList.asErrorListEnglish.T_LanguagList[92]:='Error 92';
T_ErrorList.asErrorListEnglish.T_LanguagList[93]:='Error 93';
T_ErrorList.asErrorListEnglish.T_LanguagList[94]:='Error 94';
T_ErrorList.asErrorListEnglish.T_LanguagList[95]:='Error 95';
T_ErrorList.asErrorListEnglish.T_LanguagList[96]:='Error 96';
T_ErrorList.asErrorListEnglish.T_LanguagList[97]:='Error 97';
T_ErrorList.asErrorListEnglish.T_LanguagList[98]:='USB-Stick not founded for Profile read/write';
T_ErrorList.asErrorListEnglish.T_LanguagList[99]:='USB-Stick not founded for Profile delete';
T_ErrorList.asErrorListEnglish.T_LanguagList[100]:='Power Supply is switched off';
T_ErrorList.asErrorListEnglish.T_LanguagList[101]:='At least one Profle has a syntax Error during reading of all Profiles';
T_ErrorList.asErrorListEnglish.T_LanguagList[102]:='NovRAM store failure';
T_ErrorList.asErrorListEnglish.T_LanguagList[103]:='Not handled undefined Process Error';
T_ErrorList.asErrorListEnglish.T_LanguagList[104]:='USB-Stick not founded';
T_ErrorList.asErrorListEnglish.T_LanguagList[105]:='Cylinder function not implemented';
T_ErrorList.asErrorListEnglish.T_LanguagList[106]:='Cylinder Active-->Sensor not ON';
T_ErrorList.asErrorListEnglish.T_LanguagList[107]:='Cylinder Inactive-->Sensor not ON';
T_ErrorList.asErrorListEnglish.T_LanguagList[108]:='Not handled undefined Cylinder Error';
T_ErrorList.asErrorListEnglish.T_LanguagList[109]:='Axis Brake Active of ST1';
T_ErrorList.asErrorListEnglish.T_LanguagList[110]:='Error 110';
T_ErrorList.asErrorListEnglish.T_LanguagList[111]:='Error 111';
T_ErrorList.asErrorListEnglish.T_LanguagList[112]:='Error 112';
T_ErrorList.asErrorListEnglish.T_LanguagList[113]:='Error 113';
T_ErrorList.asErrorListEnglish.T_LanguagList[114]:='Error 114';
T_ErrorList.asErrorListEnglish.T_LanguagList[115]:='Error 115';
T_ErrorList.asErrorListEnglish.T_LanguagList[116]:='Error 116';
T_ErrorList.asErrorListEnglish.T_LanguagList[117]:='Error 117';
T_ErrorList.asErrorListEnglish.T_LanguagList[118]:='Error 118';
T_ErrorList.asErrorListEnglish.T_LanguagList[119]:='Error 119';
T_ErrorList.asErrorListEnglish.T_LanguagList[120]:='Error 120';
T_ErrorList.asErrorListEnglish.T_LanguagList[121]:='Error 121';
T_ErrorList.asErrorListEnglish.T_LanguagList[122]:='Error 122';
T_ErrorList.asErrorListEnglish.T_LanguagList[123]:='Error 123';
T_ErrorList.asErrorListEnglish.T_LanguagList[124]:='Error 124';
T_ErrorList.asErrorListEnglish.T_LanguagList[125]:='Error 125';
T_ErrorList.asErrorListEnglish.T_LanguagList[126]:='Error 126';
T_ErrorList.asErrorListEnglish.T_LanguagList[127]:='Error 127';
T_ErrorList.asErrorListEnglish.T_LanguagList[128]:='Error 128';
T_ErrorList.asErrorListEnglish.T_LanguagList[129]:='Error 129';
T_ErrorList.asErrorListEnglish.T_LanguagList[130]:='Error 130';
T_ErrorList.asErrorListEnglish.T_LanguagList[131]:='Error 131';
T_ErrorList.asErrorListEnglish.T_LanguagList[132]:='Error 132';
T_ErrorList.asErrorListEnglish.T_LanguagList[133]:='Error 133';
T_ErrorList.asErrorListEnglish.T_LanguagList[134]:='Error 134';
T_ErrorList.asErrorListEnglish.T_LanguagList[135]:='Error 135';
T_ErrorList.asErrorListEnglish.T_LanguagList[136]:='Error 136';
T_ErrorList.asErrorListEnglish.T_LanguagList[137]:='Error 137';
T_ErrorList.asErrorListEnglish.T_LanguagList[138]:='Error 138';
T_ErrorList.asErrorListEnglish.T_LanguagList[139]:='Error 139';
T_ErrorList.asErrorListEnglish.T_LanguagList[140]:='Error 140';
T_ErrorList.asErrorListEnglish.T_LanguagList[141]:='Error 141';
T_ErrorList.asErrorListEnglish.T_LanguagList[142]:='Error 142';
T_ErrorList.asErrorListEnglish.T_LanguagList[143]:='Error 143';
T_ErrorList.asErrorListEnglish.T_LanguagList[144]:='Error 144';
T_ErrorList.asErrorListEnglish.T_LanguagList[145]:='Error 145';
T_ErrorList.asErrorListEnglish.T_LanguagList[146]:='HDD not Ready';
T_ErrorList.asErrorListEnglish.T_LanguagList[147]:='Timeout while write on USB-Stick';
T_ErrorList.asErrorListEnglish.T_LanguagList[148]:='USB Stick no writing';
T_ErrorList.asErrorListEnglish.T_LanguagList[149]:='USB Stick not found';
T_ErrorList.asErrorListEnglish.T_LanguagList[150]:='Error 150';
T_ErrorList.asErrorListEnglish.T_LanguagList[151]:='Error 151';
T_ErrorList.asErrorListEnglish.T_LanguagList[152]:='Error 152';
T_ErrorList.asErrorListEnglish.T_LanguagList[153]:='Error 153';
T_ErrorList.asErrorListEnglish.T_LanguagList[154]:='Error 154';
T_ErrorList.asErrorListEnglish.T_LanguagList[155]:='Error 155';
T_ErrorList.asErrorListEnglish.T_LanguagList[156]:='Error 156';
T_ErrorList.asErrorListEnglish.T_LanguagList[157]:='Error 157';
T_ErrorList.asErrorListEnglish.T_LanguagList[158]:='Error 158';
T_ErrorList.asErrorListEnglish.T_LanguagList[159]:='Error 159';
T_ErrorList.asErrorListEnglish.T_LanguagList[160]:='Error 160';
T_ErrorList.asErrorListEnglish.T_LanguagList[161]:='Error 161';
T_ErrorList.asErrorListEnglish.T_LanguagList[162]:='Error 162';
T_ErrorList.asErrorListEnglish.T_LanguagList[163]:='Error 163';
T_ErrorList.asErrorListEnglish.T_LanguagList[164]:='Error 164';
T_ErrorList.asErrorListEnglish.T_LanguagList[165]:='Error 165';
T_ErrorList.asErrorListEnglish.T_LanguagList[166]:='Error 166';
T_ErrorList.asErrorListEnglish.T_LanguagList[167]:='Error 167';
T_ErrorList.asErrorListEnglish.T_LanguagList[168]:='Error 168';
T_ErrorList.asErrorListEnglish.T_LanguagList[169]:='Error 169';
T_ErrorList.asErrorListEnglish.T_LanguagList[170]:='Error 170';
T_ErrorList.asErrorListEnglish.T_LanguagList[171]:='Error 171';
T_ErrorList.asErrorListEnglish.T_LanguagList[172]:='Error 172';
T_ErrorList.asErrorListEnglish.T_LanguagList[173]:='Error 173';
T_ErrorList.asErrorListEnglish.T_LanguagList[174]:='Error 174';
T_ErrorList.asErrorListEnglish.T_LanguagList[175]:='Error 175';
T_ErrorList.asErrorListEnglish.T_LanguagList[176]:='Error 176';
T_ErrorList.asErrorListEnglish.T_LanguagList[177]:='Error 177';
T_ErrorList.asErrorListEnglish.T_LanguagList[178]:='Error 178';
T_ErrorList.asErrorListEnglish.T_LanguagList[179]:='Error 179';
T_ErrorList.asErrorListEnglish.T_LanguagList[180]:='Error 180';
T_ErrorList.asErrorListEnglish.T_LanguagList[181]:='Error 181';
T_ErrorList.asErrorListEnglish.T_LanguagList[182]:='Error 182';
T_ErrorList.asErrorListEnglish.T_LanguagList[183]:='Error 183';
T_ErrorList.asErrorListEnglish.T_LanguagList[184]:='Error 184';
T_ErrorList.asErrorListEnglish.T_LanguagList[185]:='Error 185';
T_ErrorList.asErrorListEnglish.T_LanguagList[186]:='Error 186';
T_ErrorList.asErrorListEnglish.T_LanguagList[187]:='Error 187';
T_ErrorList.asErrorListEnglish.T_LanguagList[188]:='Error 188';
T_ErrorList.asErrorListEnglish.T_LanguagList[189]:='Error 189';
T_ErrorList.asErrorListEnglish.T_LanguagList[190]:='Error 190';
T_ErrorList.asErrorListEnglish.T_LanguagList[191]:='Error 191';
T_ErrorList.asErrorListEnglish.T_LanguagList[192]:='Error 192';
T_ErrorList.asErrorListEnglish.T_LanguagList[193]:='Error 193';
T_ErrorList.asErrorListEnglish.T_LanguagList[194]:='Error 194';
T_ErrorList.asErrorListEnglish.T_LanguagList[195]:='Error 195';
T_ErrorList.asErrorListEnglish.T_LanguagList[196]:='Error 196';
T_ErrorList.asErrorListEnglish.T_LanguagList[197]:='Error 197';
T_ErrorList.asErrorListEnglish.T_LanguagList[198]:='Error 198';
T_ErrorList.asErrorListEnglish.T_LanguagList[199]:='Error 199';
T_ErrorList.asErrorListEnglish.T_LanguagList[200]:='Error 200';
T_ErrorList.asErrorListEnglish.T_LanguagList[201]:='Error 201';
T_ErrorList.asErrorListEnglish.T_LanguagList[202]:='Error 202';
T_ErrorList.asErrorListEnglish.T_LanguagList[203]:='Error 203';
T_ErrorList.asErrorListEnglish.T_LanguagList[204]:='Error 204';
T_ErrorList.asErrorListEnglish.T_LanguagList[205]:='Error 205';
T_ErrorList.asErrorListEnglish.T_LanguagList[206]:='Error 206';
T_ErrorList.asErrorListEnglish.T_LanguagList[207]:='Error 207';
T_ErrorList.asErrorListEnglish.T_LanguagList[208]:='Error 208';
T_ErrorList.asErrorListEnglish.T_LanguagList[209]:='Error 209';
T_ErrorList.asErrorListEnglish.T_LanguagList[210]:='Error 210';
T_ErrorList.asErrorListEnglish.T_LanguagList[211]:='Error 211';
T_ErrorList.asErrorListEnglish.T_LanguagList[212]:='Error 212';
T_ErrorList.asErrorListEnglish.T_LanguagList[213]:='Error 213';
T_ErrorList.asErrorListEnglish.T_LanguagList[214]:='Error 214';
T_ErrorList.asErrorListEnglish.T_LanguagList[215]:='Error 215';
T_ErrorList.asErrorListEnglish.T_LanguagList[216]:='Error 216';
T_ErrorList.asErrorListEnglish.T_LanguagList[217]:='Error 217';
T_ErrorList.asErrorListEnglish.T_LanguagList[218]:='Error 218';
T_ErrorList.asErrorListEnglish.T_LanguagList[219]:='Error 219';
T_ErrorList.asErrorListEnglish.T_LanguagList[220]:='Error 220';
T_ErrorList.asErrorListEnglish.T_LanguagList[221]:='Error 221';
T_ErrorList.asErrorListEnglish.T_LanguagList[222]:='Error 222';
T_ErrorList.asErrorListEnglish.T_LanguagList[223]:='Error 223';
T_ErrorList.asErrorListEnglish.T_LanguagList[224]:='Error 224';
T_ErrorList.asErrorListEnglish.T_LanguagList[225]:='Error 225';
T_ErrorList.asErrorListEnglish.T_LanguagList[226]:='Error 226';
T_ErrorList.asErrorListEnglish.T_LanguagList[227]:='Error 227';
T_ErrorList.asErrorListEnglish.T_LanguagList[228]:='Error 228';
T_ErrorList.asErrorListEnglish.T_LanguagList[229]:='Error 229';
T_ErrorList.asErrorListEnglish.T_LanguagList[230]:='Error 230';
T_ErrorList.asErrorListEnglish.T_LanguagList[231]:='Error 231';
T_ErrorList.asErrorListEnglish.T_LanguagList[232]:='Error 232';
T_ErrorList.asErrorListEnglish.T_LanguagList[233]:='Error 233';
T_ErrorList.asErrorListEnglish.T_LanguagList[234]:='Error 234';
T_ErrorList.asErrorListEnglish.T_LanguagList[235]:='Error 235';
T_ErrorList.asErrorListEnglish.T_LanguagList[236]:='Error 236';
T_ErrorList.asErrorListEnglish.T_LanguagList[237]:='Error 237';
T_ErrorList.asErrorListEnglish.T_LanguagList[238]:='Error 238';
T_ErrorList.asErrorListEnglish.T_LanguagList[239]:='Error 239';
T_ErrorList.asErrorListEnglish.T_LanguagList[240]:='Error 240';
T_ErrorList.asErrorListEnglish.T_LanguagList[241]:='Error 241';
T_ErrorList.asErrorListEnglish.T_LanguagList[242]:='Error 242';
T_ErrorList.asErrorListEnglish.T_LanguagList[243]:='Error 243';
T_ErrorList.asErrorListEnglish.T_LanguagList[244]:='Error 244';
T_ErrorList.asErrorListEnglish.T_LanguagList[245]:='Error 245';
T_ErrorList.asErrorListEnglish.T_LanguagList[246]:='Error 246';
T_ErrorList.asErrorListEnglish.T_LanguagList[247]:='Error 247';
T_ErrorList.asErrorListEnglish.T_LanguagList[248]:='Error 248';
T_ErrorList.asErrorListEnglish.T_LanguagList[249]:='Error 249';
T_ErrorList.asErrorListEnglish.T_LanguagList[250]:='Error 250';
T_ErrorList.asErrorListEnglish.T_LanguagList[251]:='Error 251';
T_ErrorList.asErrorListEnglish.T_LanguagList[252]:='Error 252';
T_ErrorList.asErrorListEnglish.T_LanguagList[253]:='Error 253';
T_ErrorList.asErrorListEnglish.T_LanguagList[254]:='Error 254';
T_ErrorList.asErrorListEnglish.T_LanguagList[255]:='Error 255';
T_ErrorList.asErrorListEnglish.T_LanguagList[256]:='Error 256';
T_ErrorList.asErrorListEnglish.T_LanguagList[257]:='Error 257';
T_ErrorList.asErrorListEnglish.T_LanguagList[258]:='Error 258';
T_ErrorList.asErrorListEnglish.T_LanguagList[259]:='Error 259';
T_ErrorList.asErrorListEnglish.T_LanguagList[260]:='Error 260';
T_ErrorList.asErrorListEnglish.T_LanguagList[261]:='Error 261';
T_ErrorList.asErrorListEnglish.T_LanguagList[262]:='Error 262';
T_ErrorList.asErrorListEnglish.T_LanguagList[263]:='Error 263';
T_ErrorList.asErrorListEnglish.T_LanguagList[264]:='Error 264';
T_ErrorList.asErrorListEnglish.T_LanguagList[265]:='Error 265';
T_ErrorList.asErrorListEnglish.T_LanguagList[266]:='Error 266';
T_ErrorList.asErrorListEnglish.T_LanguagList[267]:='Error 267';
T_ErrorList.asErrorListEnglish.T_LanguagList[268]:='Error 268';
T_ErrorList.asErrorListEnglish.T_LanguagList[269]:='Error 269';
T_ErrorList.asErrorListEnglish.T_LanguagList[270]:='Error 270';
T_ErrorList.asErrorListEnglish.T_LanguagList[271]:='Error 271';
T_ErrorList.asErrorListEnglish.T_LanguagList[272]:='Error 272';
T_ErrorList.asErrorListEnglish.T_LanguagList[273]:='Error 273';
T_ErrorList.asErrorListEnglish.T_LanguagList[274]:='Error 274';
T_ErrorList.asErrorListEnglish.T_LanguagList[275]:='Error 275';
T_ErrorList.asErrorListEnglish.T_LanguagList[276]:='Error 276';
T_ErrorList.asErrorListEnglish.T_LanguagList[277]:='Error 277';
T_ErrorList.asErrorListEnglish.T_LanguagList[278]:='Error 278';
T_ErrorList.asErrorListEnglish.T_LanguagList[279]:='Error 279';
T_ErrorList.asErrorListEnglish.T_LanguagList[280]:='Error 280';
T_ErrorList.asErrorListEnglish.T_LanguagList[281]:='Error 281';
T_ErrorList.asErrorListEnglish.T_LanguagList[282]:='Error 282';
T_ErrorList.asErrorListEnglish.T_LanguagList[283]:='Error 283';
T_ErrorList.asErrorListEnglish.T_LanguagList[284]:='Error 284';
T_ErrorList.asErrorListEnglish.T_LanguagList[285]:='Error 285';
T_ErrorList.asErrorListEnglish.T_LanguagList[286]:='Error 286';
T_ErrorList.asErrorListEnglish.T_LanguagList[287]:='Error 287';
T_ErrorList.asErrorListEnglish.T_LanguagList[288]:='Error 288';
T_ErrorList.asErrorListEnglish.T_LanguagList[289]:='Error 289';
T_ErrorList.asErrorListEnglish.T_LanguagList[290]:='Error 290';
T_ErrorList.asErrorListEnglish.T_LanguagList[291]:='Error 291';
T_ErrorList.asErrorListEnglish.T_LanguagList[292]:='Error 292';
T_ErrorList.asErrorListEnglish.T_LanguagList[293]:='Error 293';
T_ErrorList.asErrorListEnglish.T_LanguagList[294]:='Error 294';
T_ErrorList.asErrorListEnglish.T_LanguagList[295]:='Error 295';
T_ErrorList.asErrorListEnglish.T_LanguagList[296]:='Error 296';
T_ErrorList.asErrorListEnglish.T_LanguagList[297]:='Error 297';
T_ErrorList.asErrorListEnglish.T_LanguagList[298]:='Error 298';
T_ErrorList.asErrorListEnglish.T_LanguagList[299]:='Error 299';
T_ErrorList.asErrorListEnglish.T_LanguagList[300]:='Error 300';

(* Static Francais Error List *)
T_ErrorList.asErrorListFrancais.T_LanguagList[1]:='Error 1';
T_ErrorList.asErrorListFrancais.T_LanguagList[2]:='Error 2';
T_ErrorList.asErrorListFrancais.T_LanguagList[3]:='Error 3';
T_ErrorList.asErrorListFrancais.T_LanguagList[4]:='Error 4';
T_ErrorList.asErrorListFrancais.T_LanguagList[5]:='Error 5';
T_ErrorList.asErrorListFrancais.T_LanguagList[6]:='Error 6';
T_ErrorList.asErrorListFrancais.T_LanguagList[7]:='Error 7';
T_ErrorList.asErrorListFrancais.T_LanguagList[8]:='Error 8';
T_ErrorList.asErrorListFrancais.T_LanguagList[9]:='Error 9';
T_ErrorList.asErrorListFrancais.T_LanguagList[10]:='Error 10';
T_ErrorList.asErrorListFrancais.T_LanguagList[11]:='Error 11';
T_ErrorList.asErrorListFrancais.T_LanguagList[12]:='Error 12';
T_ErrorList.asErrorListFrancais.T_LanguagList[13]:='Error 13';
T_ErrorList.asErrorListFrancais.T_LanguagList[14]:='Error 14';
T_ErrorList.asErrorListFrancais.T_LanguagList[15]:='Error 15';
T_ErrorList.asErrorListFrancais.T_LanguagList[16]:='Error 16';
T_ErrorList.asErrorListFrancais.T_LanguagList[17]:='Error 17';
T_ErrorList.asErrorListFrancais.T_LanguagList[18]:='Error 18';
T_ErrorList.asErrorListFrancais.T_LanguagList[19]:='Error 19';
T_ErrorList.asErrorListFrancais.T_LanguagList[20]:='Error 20';
T_ErrorList.asErrorListFrancais.T_LanguagList[21]:='Error 21';
T_ErrorList.asErrorListFrancais.T_LanguagList[22]:='Error 22';
T_ErrorList.asErrorListFrancais.T_LanguagList[23]:='Error 23';
T_ErrorList.asErrorListFrancais.T_LanguagList[24]:='Error 24';
T_ErrorList.asErrorListFrancais.T_LanguagList[25]:='Error 25';
T_ErrorList.asErrorListFrancais.T_LanguagList[26]:='Error 26';
T_ErrorList.asErrorListFrancais.T_LanguagList[27]:='Error 27';
T_ErrorList.asErrorListFrancais.T_LanguagList[28]:='Error 28';
T_ErrorList.asErrorListFrancais.T_LanguagList[29]:='Error 29';
T_ErrorList.asErrorListFrancais.T_LanguagList[30]:='Error 30';
T_ErrorList.asErrorListFrancais.T_LanguagList[31]:='Error 31';
T_ErrorList.asErrorListFrancais.T_LanguagList[32]:='Error 32';
T_ErrorList.asErrorListFrancais.T_LanguagList[33]:='Error 33';
T_ErrorList.asErrorListFrancais.T_LanguagList[34]:='Error 34';
T_ErrorList.asErrorListFrancais.T_LanguagList[35]:='Error 35';
T_ErrorList.asErrorListFrancais.T_LanguagList[36]:='Error 36';
T_ErrorList.asErrorListFrancais.T_LanguagList[37]:='Error 37';
T_ErrorList.asErrorListFrancais.T_LanguagList[38]:='Error 38';
T_ErrorList.asErrorListFrancais.T_LanguagList[39]:='Error 39';
T_ErrorList.asErrorListFrancais.T_LanguagList[40]:='Error 40';
T_ErrorList.asErrorListFrancais.T_LanguagList[41]:='Error 41';
T_ErrorList.asErrorListFrancais.T_LanguagList[42]:='Error 42';
T_ErrorList.asErrorListFrancais.T_LanguagList[43]:='Error 43';
T_ErrorList.asErrorListFrancais.T_LanguagList[44]:='Error 44';
T_ErrorList.asErrorListFrancais.T_LanguagList[45]:='Error 45';
T_ErrorList.asErrorListFrancais.T_LanguagList[46]:='Error 46';
T_ErrorList.asErrorListFrancais.T_LanguagList[47]:='Error 47';
T_ErrorList.asErrorListFrancais.T_LanguagList[48]:='Error 48';
T_ErrorList.asErrorListFrancais.T_LanguagList[49]:='Error 49';
T_ErrorList.asErrorListFrancais.T_LanguagList[50]:='Error 50';
T_ErrorList.asErrorListFrancais.T_LanguagList[51]:='Error 51';
T_ErrorList.asErrorListFrancais.T_LanguagList[52]:='Error 52';
T_ErrorList.asErrorListFrancais.T_LanguagList[53]:='Error 53';
T_ErrorList.asErrorListFrancais.T_LanguagList[54]:='Error 54';
T_ErrorList.asErrorListFrancais.T_LanguagList[55]:='Error 55';
T_ErrorList.asErrorListFrancais.T_LanguagList[56]:='Error 56';
T_ErrorList.asErrorListFrancais.T_LanguagList[57]:='Error 57';
T_ErrorList.asErrorListFrancais.T_LanguagList[58]:='Error 58';
T_ErrorList.asErrorListFrancais.T_LanguagList[59]:='Error 59';
T_ErrorList.asErrorListFrancais.T_LanguagList[60]:='Error 60';
T_ErrorList.asErrorListFrancais.T_LanguagList[61]:='Error 61';
T_ErrorList.asErrorListFrancais.T_LanguagList[62]:='Error 62';
T_ErrorList.asErrorListFrancais.T_LanguagList[63]:='Error 63';
T_ErrorList.asErrorListFrancais.T_LanguagList[64]:='Error 64';
T_ErrorList.asErrorListFrancais.T_LanguagList[65]:='Error 65';
T_ErrorList.asErrorListFrancais.T_LanguagList[66]:='Error 66';
T_ErrorList.asErrorListFrancais.T_LanguagList[67]:='Error 67';
T_ErrorList.asErrorListFrancais.T_LanguagList[68]:='Error 68';
T_ErrorList.asErrorListFrancais.T_LanguagList[69]:='Error 69';
T_ErrorList.asErrorListFrancais.T_LanguagList[70]:='Error 70';
T_ErrorList.asErrorListFrancais.T_LanguagList[71]:='Error 71';
T_ErrorList.asErrorListFrancais.T_LanguagList[72]:='Error 72';
T_ErrorList.asErrorListFrancais.T_LanguagList[73]:='Error 73';
T_ErrorList.asErrorListFrancais.T_LanguagList[74]:='Error 74';
T_ErrorList.asErrorListFrancais.T_LanguagList[75]:='Error 75';
T_ErrorList.asErrorListFrancais.T_LanguagList[76]:='Error 76';
T_ErrorList.asErrorListFrancais.T_LanguagList[77]:='Error 77';
T_ErrorList.asErrorListFrancais.T_LanguagList[78]:='Error 78';
T_ErrorList.asErrorListFrancais.T_LanguagList[79]:='Error 79';
T_ErrorList.asErrorListFrancais.T_LanguagList[80]:='Error 80';
T_ErrorList.asErrorListFrancais.T_LanguagList[81]:='Error 81';
T_ErrorList.asErrorListFrancais.T_LanguagList[82]:='Error 82';
T_ErrorList.asErrorListFrancais.T_LanguagList[83]:='Error 83';
T_ErrorList.asErrorListFrancais.T_LanguagList[84]:='Error 84';
T_ErrorList.asErrorListFrancais.T_LanguagList[85]:='Error 85';
T_ErrorList.asErrorListFrancais.T_LanguagList[86]:='Error 86';
T_ErrorList.asErrorListFrancais.T_LanguagList[87]:='Error 87';
T_ErrorList.asErrorListFrancais.T_LanguagList[88]:='Error 88';
T_ErrorList.asErrorListFrancais.T_LanguagList[89]:='Error 89';
T_ErrorList.asErrorListFrancais.T_LanguagList[90]:='Error 90';
T_ErrorList.asErrorListFrancais.T_LanguagList[91]:='Error 91';
T_ErrorList.asErrorListFrancais.T_LanguagList[92]:='Error 92';
T_ErrorList.asErrorListFrancais.T_LanguagList[93]:='Error 93';
T_ErrorList.asErrorListFrancais.T_LanguagList[94]:='Error 94';
T_ErrorList.asErrorListFrancais.T_LanguagList[95]:='Error 95';
T_ErrorList.asErrorListFrancais.T_LanguagList[96]:='Error 96';
T_ErrorList.asErrorListFrancais.T_LanguagList[97]:='Error 97';
T_ErrorList.asErrorListFrancais.T_LanguagList[98]:='Error 98';
T_ErrorList.asErrorListFrancais.T_LanguagList[99]:='Error 99';
T_ErrorList.asErrorListFrancais.T_LanguagList[100]:='Error 100';
T_ErrorList.asErrorListFrancais.T_LanguagList[101]:='Error 101';
T_ErrorList.asErrorListFrancais.T_LanguagList[102]:='Error 102';
T_ErrorList.asErrorListFrancais.T_LanguagList[103]:='Error 103';
T_ErrorList.asErrorListFrancais.T_LanguagList[104]:='Error 104';
T_ErrorList.asErrorListFrancais.T_LanguagList[105]:='Error 105';
T_ErrorList.asErrorListFrancais.T_LanguagList[106]:='Error 106';
T_ErrorList.asErrorListFrancais.T_LanguagList[107]:='Error 107';
T_ErrorList.asErrorListFrancais.T_LanguagList[108]:='Error 108';
T_ErrorList.asErrorListFrancais.T_LanguagList[109]:='Error 109';
T_ErrorList.asErrorListFrancais.T_LanguagList[110]:='Error 110';
T_ErrorList.asErrorListFrancais.T_LanguagList[111]:='Error 111';
T_ErrorList.asErrorListFrancais.T_LanguagList[112]:='Error 112';
T_ErrorList.asErrorListFrancais.T_LanguagList[113]:='Error 113';
T_ErrorList.asErrorListFrancais.T_LanguagList[114]:='Error 114';
T_ErrorList.asErrorListFrancais.T_LanguagList[115]:='Error 115';
T_ErrorList.asErrorListFrancais.T_LanguagList[116]:='Error 116';
T_ErrorList.asErrorListFrancais.T_LanguagList[117]:='Error 117';
T_ErrorList.asErrorListFrancais.T_LanguagList[118]:='Error 118';
T_ErrorList.asErrorListFrancais.T_LanguagList[119]:='Error 119';
T_ErrorList.asErrorListFrancais.T_LanguagList[120]:='Error 120';
T_ErrorList.asErrorListFrancais.T_LanguagList[121]:='Error 121';
T_ErrorList.asErrorListFrancais.T_LanguagList[122]:='Error 122';
T_ErrorList.asErrorListFrancais.T_LanguagList[123]:='Error 123';
T_ErrorList.asErrorListFrancais.T_LanguagList[124]:='Error 124';
T_ErrorList.asErrorListFrancais.T_LanguagList[125]:='Error 125';
T_ErrorList.asErrorListFrancais.T_LanguagList[126]:='Error 126';
T_ErrorList.asErrorListFrancais.T_LanguagList[127]:='Error 127';
T_ErrorList.asErrorListFrancais.T_LanguagList[128]:='Error 128';
T_ErrorList.asErrorListFrancais.T_LanguagList[129]:='Error 129';
T_ErrorList.asErrorListFrancais.T_LanguagList[130]:='Error 130';
T_ErrorList.asErrorListFrancais.T_LanguagList[131]:='Error 131';
T_ErrorList.asErrorListFrancais.T_LanguagList[132]:='Error 132';
T_ErrorList.asErrorListFrancais.T_LanguagList[133]:='Error 133';
T_ErrorList.asErrorListFrancais.T_LanguagList[134]:='Error 134';
T_ErrorList.asErrorListFrancais.T_LanguagList[135]:='Error 135';
T_ErrorList.asErrorListFrancais.T_LanguagList[136]:='Error 136';
T_ErrorList.asErrorListFrancais.T_LanguagList[137]:='Error 137';
T_ErrorList.asErrorListFrancais.T_LanguagList[138]:='Error 138';
T_ErrorList.asErrorListFrancais.T_LanguagList[139]:='Error 139';
T_ErrorList.asErrorListFrancais.T_LanguagList[140]:='Error 140';
T_ErrorList.asErrorListFrancais.T_LanguagList[141]:='Error 141';
T_ErrorList.asErrorListFrancais.T_LanguagList[142]:='Error 142';
T_ErrorList.asErrorListFrancais.T_LanguagList[143]:='Error 143';
T_ErrorList.asErrorListFrancais.T_LanguagList[144]:='Error 144';
T_ErrorList.asErrorListFrancais.T_LanguagList[145]:='Error 145';
T_ErrorList.asErrorListFrancais.T_LanguagList[146]:='Error 146';
T_ErrorList.asErrorListFrancais.T_LanguagList[147]:='Error 147';
T_ErrorList.asErrorListFrancais.T_LanguagList[148]:='Error 148';
T_ErrorList.asErrorListFrancais.T_LanguagList[149]:='Error 149';
T_ErrorList.asErrorListFrancais.T_LanguagList[150]:='Error 150';
T_ErrorList.asErrorListFrancais.T_LanguagList[151]:='Error 151';
T_ErrorList.asErrorListFrancais.T_LanguagList[152]:='Error 152';
T_ErrorList.asErrorListFrancais.T_LanguagList[153]:='Error 153';
T_ErrorList.asErrorListFrancais.T_LanguagList[154]:='Error 154';
T_ErrorList.asErrorListFrancais.T_LanguagList[155]:='Error 155';
T_ErrorList.asErrorListFrancais.T_LanguagList[156]:='Error 156';
T_ErrorList.asErrorListFrancais.T_LanguagList[157]:='Error 157';
T_ErrorList.asErrorListFrancais.T_LanguagList[158]:='Error 158';
T_ErrorList.asErrorListFrancais.T_LanguagList[159]:='Error 159';
T_ErrorList.asErrorListFrancais.T_LanguagList[160]:='Error 160';
T_ErrorList.asErrorListFrancais.T_LanguagList[161]:='Error 161';
T_ErrorList.asErrorListFrancais.T_LanguagList[162]:='Error 162';
T_ErrorList.asErrorListFrancais.T_LanguagList[163]:='Error 163';
T_ErrorList.asErrorListFrancais.T_LanguagList[164]:='Error 164';
T_ErrorList.asErrorListFrancais.T_LanguagList[165]:='Error 165';
T_ErrorList.asErrorListFrancais.T_LanguagList[166]:='Error 166';
T_ErrorList.asErrorListFrancais.T_LanguagList[167]:='Error 167';
T_ErrorList.asErrorListFrancais.T_LanguagList[168]:='Error 168';
T_ErrorList.asErrorListFrancais.T_LanguagList[169]:='Error 169';
T_ErrorList.asErrorListFrancais.T_LanguagList[170]:='Error 170';
T_ErrorList.asErrorListFrancais.T_LanguagList[171]:='Error 171';
T_ErrorList.asErrorListFrancais.T_LanguagList[172]:='Error 172';
T_ErrorList.asErrorListFrancais.T_LanguagList[173]:='Error 173';
T_ErrorList.asErrorListFrancais.T_LanguagList[174]:='Error 174';
T_ErrorList.asErrorListFrancais.T_LanguagList[175]:='Error 175';
T_ErrorList.asErrorListFrancais.T_LanguagList[176]:='Error 176';
T_ErrorList.asErrorListFrancais.T_LanguagList[177]:='Error 177';
T_ErrorList.asErrorListFrancais.T_LanguagList[178]:='Error 178';
T_ErrorList.asErrorListFrancais.T_LanguagList[179]:='Error 179';
T_ErrorList.asErrorListFrancais.T_LanguagList[180]:='Error 180';
T_ErrorList.asErrorListFrancais.T_LanguagList[181]:='Error 181';
T_ErrorList.asErrorListFrancais.T_LanguagList[182]:='Error 182';
T_ErrorList.asErrorListFrancais.T_LanguagList[183]:='Error 183';
T_ErrorList.asErrorListFrancais.T_LanguagList[184]:='Error 184';
T_ErrorList.asErrorListFrancais.T_LanguagList[185]:='Error 185';
T_ErrorList.asErrorListFrancais.T_LanguagList[186]:='Error 186';
T_ErrorList.asErrorListFrancais.T_LanguagList[187]:='Error 187';
T_ErrorList.asErrorListFrancais.T_LanguagList[188]:='Error 188';
T_ErrorList.asErrorListFrancais.T_LanguagList[189]:='Error 189';
T_ErrorList.asErrorListFrancais.T_LanguagList[190]:='Error 190';
T_ErrorList.asErrorListFrancais.T_LanguagList[191]:='Error 191';
T_ErrorList.asErrorListFrancais.T_LanguagList[192]:='Error 192';
T_ErrorList.asErrorListFrancais.T_LanguagList[193]:='Error 193';
T_ErrorList.asErrorListFrancais.T_LanguagList[194]:='Error 194';
T_ErrorList.asErrorListFrancais.T_LanguagList[195]:='Error 195';
T_ErrorList.asErrorListFrancais.T_LanguagList[196]:='Error 196';
T_ErrorList.asErrorListFrancais.T_LanguagList[197]:='Error 197';
T_ErrorList.asErrorListFrancais.T_LanguagList[198]:='Error 198';
T_ErrorList.asErrorListFrancais.T_LanguagList[199]:='Error 199';
T_ErrorList.asErrorListFrancais.T_LanguagList[200]:='Error 200';
T_ErrorList.asErrorListFrancais.T_LanguagList[201]:='Error 201';
T_ErrorList.asErrorListFrancais.T_LanguagList[202]:='Error 202';
T_ErrorList.asErrorListFrancais.T_LanguagList[203]:='Error 203';
T_ErrorList.asErrorListFrancais.T_LanguagList[204]:='Error 204';
T_ErrorList.asErrorListFrancais.T_LanguagList[205]:='Error 205';
T_ErrorList.asErrorListFrancais.T_LanguagList[206]:='Error 206';
T_ErrorList.asErrorListFrancais.T_LanguagList[207]:='Error 207';
T_ErrorList.asErrorListFrancais.T_LanguagList[208]:='Error 208';
T_ErrorList.asErrorListFrancais.T_LanguagList[209]:='Error 209';
T_ErrorList.asErrorListFrancais.T_LanguagList[210]:='Error 210';
T_ErrorList.asErrorListFrancais.T_LanguagList[211]:='Error 211';
T_ErrorList.asErrorListFrancais.T_LanguagList[212]:='Error 212';
T_ErrorList.asErrorListFrancais.T_LanguagList[213]:='Error 213';
T_ErrorList.asErrorListFrancais.T_LanguagList[214]:='Error 214';
T_ErrorList.asErrorListFrancais.T_LanguagList[215]:='Error 215';
T_ErrorList.asErrorListFrancais.T_LanguagList[216]:='Error 216';
T_ErrorList.asErrorListFrancais.T_LanguagList[217]:='Error 217';
T_ErrorList.asErrorListFrancais.T_LanguagList[218]:='Error 218';
T_ErrorList.asErrorListFrancais.T_LanguagList[219]:='Error 219';
T_ErrorList.asErrorListFrancais.T_LanguagList[220]:='Error 220';
T_ErrorList.asErrorListFrancais.T_LanguagList[221]:='Error 221';
T_ErrorList.asErrorListFrancais.T_LanguagList[222]:='Error 222';
T_ErrorList.asErrorListFrancais.T_LanguagList[223]:='Error 223';
T_ErrorList.asErrorListFrancais.T_LanguagList[224]:='Error 224';
T_ErrorList.asErrorListFrancais.T_LanguagList[225]:='Error 225';
T_ErrorList.asErrorListFrancais.T_LanguagList[226]:='Error 226';
T_ErrorList.asErrorListFrancais.T_LanguagList[227]:='Error 227';
T_ErrorList.asErrorListFrancais.T_LanguagList[228]:='Error 228';
T_ErrorList.asErrorListFrancais.T_LanguagList[229]:='Error 229';
T_ErrorList.asErrorListFrancais.T_LanguagList[230]:='Error 230';
T_ErrorList.asErrorListFrancais.T_LanguagList[231]:='Error 231';
T_ErrorList.asErrorListFrancais.T_LanguagList[232]:='Error 232';
T_ErrorList.asErrorListFrancais.T_LanguagList[233]:='Error 233';
T_ErrorList.asErrorListFrancais.T_LanguagList[234]:='Error 234';
T_ErrorList.asErrorListFrancais.T_LanguagList[235]:='Error 235';
T_ErrorList.asErrorListFrancais.T_LanguagList[236]:='Error 236';
T_ErrorList.asErrorListFrancais.T_LanguagList[237]:='Error 237';
T_ErrorList.asErrorListFrancais.T_LanguagList[238]:='Error 238';
T_ErrorList.asErrorListFrancais.T_LanguagList[239]:='Error 239';
T_ErrorList.asErrorListFrancais.T_LanguagList[240]:='Error 240';
T_ErrorList.asErrorListFrancais.T_LanguagList[241]:='Error 241';
T_ErrorList.asErrorListFrancais.T_LanguagList[242]:='Error 242';
T_ErrorList.asErrorListFrancais.T_LanguagList[243]:='Error 243';
T_ErrorList.asErrorListFrancais.T_LanguagList[244]:='Error 244';
T_ErrorList.asErrorListFrancais.T_LanguagList[245]:='Error 245';
T_ErrorList.asErrorListFrancais.T_LanguagList[246]:='Error 246';
T_ErrorList.asErrorListFrancais.T_LanguagList[247]:='Error 247';
T_ErrorList.asErrorListFrancais.T_LanguagList[248]:='Error 248';
T_ErrorList.asErrorListFrancais.T_LanguagList[249]:='Error 249';
T_ErrorList.asErrorListFrancais.T_LanguagList[250]:='Error 250';
T_ErrorList.asErrorListFrancais.T_LanguagList[251]:='Error 251';
T_ErrorList.asErrorListFrancais.T_LanguagList[252]:='Error 252';
T_ErrorList.asErrorListFrancais.T_LanguagList[253]:='Error 253';
T_ErrorList.asErrorListFrancais.T_LanguagList[254]:='Error 254';
T_ErrorList.asErrorListFrancais.T_LanguagList[255]:='Error 255';
T_ErrorList.asErrorListFrancais.T_LanguagList[256]:='Error 256';
T_ErrorList.asErrorListFrancais.T_LanguagList[257]:='Error 257';
T_ErrorList.asErrorListFrancais.T_LanguagList[258]:='Error 258';
T_ErrorList.asErrorListFrancais.T_LanguagList[259]:='Error 259';
T_ErrorList.asErrorListFrancais.T_LanguagList[260]:='Error 260';
T_ErrorList.asErrorListFrancais.T_LanguagList[261]:='Error 261';
T_ErrorList.asErrorListFrancais.T_LanguagList[262]:='Error 262';
T_ErrorList.asErrorListFrancais.T_LanguagList[263]:='Error 263';
T_ErrorList.asErrorListFrancais.T_LanguagList[264]:='Error 264';
T_ErrorList.asErrorListFrancais.T_LanguagList[265]:='Error 265';
T_ErrorList.asErrorListFrancais.T_LanguagList[266]:='Error 266';
T_ErrorList.asErrorListFrancais.T_LanguagList[267]:='Error 267';
T_ErrorList.asErrorListFrancais.T_LanguagList[268]:='Error 268';
T_ErrorList.asErrorListFrancais.T_LanguagList[269]:='Error 269';
T_ErrorList.asErrorListFrancais.T_LanguagList[270]:='Error 270';
T_ErrorList.asErrorListFrancais.T_LanguagList[271]:='Error 271';
T_ErrorList.asErrorListFrancais.T_LanguagList[272]:='Error 272';
T_ErrorList.asErrorListFrancais.T_LanguagList[273]:='Error 273';
T_ErrorList.asErrorListFrancais.T_LanguagList[274]:='Error 274';
T_ErrorList.asErrorListFrancais.T_LanguagList[275]:='Error 275';
T_ErrorList.asErrorListFrancais.T_LanguagList[276]:='Error 276';
T_ErrorList.asErrorListFrancais.T_LanguagList[277]:='Error 277';
T_ErrorList.asErrorListFrancais.T_LanguagList[278]:='Error 278';
T_ErrorList.asErrorListFrancais.T_LanguagList[279]:='Error 279';
T_ErrorList.asErrorListFrancais.T_LanguagList[280]:='Error 280';
T_ErrorList.asErrorListFrancais.T_LanguagList[281]:='Error 281';
T_ErrorList.asErrorListFrancais.T_LanguagList[282]:='Error 282';
T_ErrorList.asErrorListFrancais.T_LanguagList[283]:='Error 283';
T_ErrorList.asErrorListFrancais.T_LanguagList[284]:='Error 284';
T_ErrorList.asErrorListFrancais.T_LanguagList[285]:='Error 285';
T_ErrorList.asErrorListFrancais.T_LanguagList[286]:='Error 286';
T_ErrorList.asErrorListFrancais.T_LanguagList[287]:='Error 287';
T_ErrorList.asErrorListFrancais.T_LanguagList[288]:='Error 288';
T_ErrorList.asErrorListFrancais.T_LanguagList[289]:='Error 289';
T_ErrorList.asErrorListFrancais.T_LanguagList[290]:='Error 290';
T_ErrorList.asErrorListFrancais.T_LanguagList[291]:='Error 291';
T_ErrorList.asErrorListFrancais.T_LanguagList[292]:='Error 292';
T_ErrorList.asErrorListFrancais.T_LanguagList[293]:='Error 293';
T_ErrorList.asErrorListFrancais.T_LanguagList[294]:='Error 294';
T_ErrorList.asErrorListFrancais.T_LanguagList[295]:='Error 295';
T_ErrorList.asErrorListFrancais.T_LanguagList[296]:='Error 296';
T_ErrorList.asErrorListFrancais.T_LanguagList[297]:='Error 297';
T_ErrorList.asErrorListFrancais.T_LanguagList[298]:='Error 298';
T_ErrorList.asErrorListFrancais.T_LanguagList[299]:='Error 299';
T_ErrorList.asErrorListFrancais.T_LanguagList[300]:='Error 300';
END_FUNCTION_BLOCK

(* POU GENERAL/FB_SAFETYLOGIC, ST *)
FUNCTION_BLOCK FB_SAFETYLOGIC
VAR_INPUT
	T_TwinSafeIn:ST_TWINSAFE_IN;
	T_TwinSafeOut:ST_TWINSAFE_OUT;
	xActiveBooting:BOOL;
	xVisuFunctionActive:BOOL;
	dwActualPage:DWORD;			(* activate page on the visualisation *)
	xOverlayMessageAcitve:BOOL;
	iStateMessage:INT;
	TCommonAxis : ST_AXIS;
END_VAR
VAR_IN_OUT
	xActiveBootingError:BOOL;
END_VAR
VAR_OUTPUT
	bStateSafetyCtrl:BYTE;
	xSafetyNotActive: BOOL;
END_VAR
VAR
	FBCheckSetupMode: FB_CHECKSETUPMODE;
	xNoEmergency: BOOL;
	xGeneralState: BOOL;
	xMachineDoorUpClose: BOOL;
	xMachineDoorClose: BOOL;
	xCheckStateEnableSwitch: BOOL;
	TONWaitCheck: TON;
	xGeneralEnergyON: BOOL;
END_VAR
FBCheckSetupMode(T_TwinSafeIn:=T_TwinSafeIn);

gT_SafetyStatus.iSetupMode:=					FBCheckSetupMode.iSetupMode;

gT_SafetyStatus.xSetupOperateModeActive:=		(T_TwinSafeIn.IxKeySwitchProcObservationCh1 AND T_TwinSafeIn.IxKeySwitchProcObservationCh2) OR (T_TwinSafeIn.IxKeySwitchWorkStationCh1 AND T_TwinSafeIn.IxKeySwitchWorkStationCh2);

xNoEmergency:=			T_TwinSafeIn.IxEmergencyStopButtonCh1 AND T_TwinSafeIn.IxEmergencyStopButtonCh2;

xMachineDoorUpClose:=	(T_TwinSafeIn.IxCabinDoorCloseCh1 AND T_TwinSafeIn.IxCabinDoorCloseCh2 AND T_TwinSafeIn.IxCabinDoorClose AND
						NOT(T_TwinSafeIn.IxCabinDoorOpen));

xMachineDoorClose:=					xMachineDoorUpClose;

gT_SafetyStatus.xSecurityDoorOpen:=	NOT(xMachineDoorClose);

gT_SafetyStatus.xSecurityDoorClose:=	xMachineDoorClose;

gT_SafetyStatus.xSecuritySwitch:=		T_TwinSafeIn.IxAxesCurrentOffCh1 AND T_TwinSafeIn.IxAxesCurrentOffCh2;


xGeneralEnergyON:=	T_TwinSafeOut.QxContactorMasterModul400VCh1 AND T_TwinSafeOut.QxContactorMasterModul400VCh2 AND
						T_TwinSafeOut.QxContactor24VCh1 AND T_TwinSafeOut.QxContactor24VCh2;

gT_SafetyStatus.xMachineDoorClose:=				xMachineDoorUpClose;

gT_SafetyStatus.xMachineEmergStopActive:=			NOT(xNoEmergency);

gT_SafetyStatus.xEnergyONNormalMode:=			xGeneralEnergyON AND
													T_TwinSafeOut.QxEnablingAxisSpindle_St1 AND
													IxTwinSafeQuickStopMaster1_1;

gT_SafetyStatus.xEnergyONSetupModeASt1:=		xGeneralEnergyON AND
													T_TwinSafeOut.QxEnablingAxisSpindle_St1 AND
													IxTwinSafeQuickStopMaster1_1;

gT_SafetyStatus.xEnergyONSetupModeBSt1:=		xGeneralEnergyON AND
													T_TwinSafeOut.QxEnablingAxisSpindle_St1 AND
													IxTwinSafeQuickStopMaster1_1;

xGeneralState:=	T_TwinSafeIn.IxReadyToOperateMasterModul1 AND T_TwinSafeIn.IxReadyToOperateMasterModul2;

IF NOT(gT_SafetyStatus.xSetupOperateModeActive) THEN
	xSafetyNotActive:=		xNoEmergency AND xMachineDoorUpClose AND
							NOT(T_TwinSafe_Status_Z_Axis_St1.xError) AND NOT(T_TwinSafe_Status_S2_Axis_St1.xError) AND NOT(T_TwinSafe_Status_S3_Axis_St1.xError) AND xGeneralState AND gT_SafetyStatus.xSecuritySwitch;
ELSE
	IF (gT_SafetyStatus.iSetupMode = 1)THEN
		xSafetyNotActive:=	xNoEmergency AND xGeneralState AND gT_SafetyStatus.xSecuritySwitch AND
							NOT(T_TwinSafe_Status_Z_Axis_St1.xError) AND NOT(T_TwinSafe_Status_S2_Axis_St1.xError) AND NOT(T_TwinSafe_Status_S3_Axis_St1.xError);
	ELSIF (gT_SafetyStatus.iSetupMode = 2)THEN
		xSafetyNotActive:=	xNoEmergency AND xGeneralState AND gT_SafetyStatus.xSecuritySwitch AND
							NOT(T_TwinSafe_Status_Z_Axis_St1.xError) AND NOT(T_TwinSafe_Status_S2_Axis_St1.xError) AND NOT(T_TwinSafe_Status_S3_Axis_St1.xError);
	END_IF;
END_IF;

xCheckStateEnableSwitch:=FALSE;
bStateSafetyCtrl:=99;	(* 99=Sicherheitsmeldungen unterdrücken *)
IF (dwActualPage = gT_PageNumber.iStart_Page1) OR (dwActualPage = gT_PageNumber.iBIOS_Page1) OR (dwActualPage = gT_PageNumber.iBIOS_Page2) THEN
	(* Sicherheitsmeldungen für wenn Maschine noch nicht aufgestartet ist *)
	IF NOT(xNoEmergency) THEN
		bStateSafetyCtrl:=19;	(* < Not Aus Taster Maschine deaktivieren > *)
	ELSIF NOT(gT_SafetyStatus.xSecuritySwitch) THEN
		bStateSafetyCtrl:=17;	(* < AntriebSperrTaste deaktivieren > *)
	ELSIF NOT(xOverlayMessageAcitve) AND xActiveBootingError AND (iStateMessage <> 401) THEN
		xActiveBootingError:=FALSE;
	ELSIF xOverlayMessageAcitve OR xActiveBootingError OR (iStateMessage = 401) THEN
		bStateSafetyCtrl:=99;	(* Keine Meldung Anzeigen-->Auserhalb des FB muss die Sicherheitsmeldung auf der Visualisierung unterdrückt werden *)
	ELSIF NOT(T_TwinSafeIn.IxReadyToOperateMasterModul1) THEN
		bStateSafetyCtrl:=12;	(* < Servo MasterModul 1 steht nicht bereit > *)
	ELSIF NOT(T_TwinSafeIn.IxReadyToOperateMasterModul2) THEN
		bStateSafetyCtrl:=13;	(* < Servo MasterModul 2 steht nicht bereit > *)
	ELSIF NOT(xMachineDoorUpClose) THEN
		bStateSafetyCtrl:=5;	(* < MaschinenTüre schliessen > *)
	ELSIF gT_SafetyStatus.xSetupOperateModeActive THEN
		bStateSafetyCtrl:=18; 	(* < Schlüsselschalter deaktivieren > *)
	ELSIF NOT(gT_SafetyStatus.xEnergyONNormalMode) AND QxCtrlLampReleaseButton THEN
		bStateSafetyCtrl:=2;	(* < FreigabeTaste drücken > *)
	ELSIF gT_SafetyStatus.xEnergyONNormalMode AND NOT(xActiveBooting) THEN
		bStateSafetyCtrl:=3;	(* < StartTaste drücken > *)
	ELSIF gT_SafetyStatus.xEnergyONNormalMode AND xActiveBooting THEN
		bStateSafetyCtrl:=1;	(* < Maschine ist am aufstarten... > *)
	END_IF;
ELSE
	(* Sicherheitsmeldungen für wenn Maschine aufgestartet ist *)
	IF xOverlayMessageAcitve OR (iStateMessage = 401) THEN
		bStateSafetyCtrl:=99;	(* Keine Meldung Anzeigen-->Auserhalb des FB muss die Sicherheitsmeldung auf der Visualisierung unterdrückt werden *)
	ELSIF NOT(T_TwinSafeIn.IxReadyToOperateMasterModul1) THEN
		bStateSafetyCtrl:=12;	(* < Servo MasterModul 1 steht nicht bereit > *)
	ELSIF NOT(T_TwinSafeIn.IxReadyToOperateMasterModul2) THEN
		bStateSafetyCtrl:=13;	(* < Servo MasterModul 2 steht nicht bereit > *)
	ELSE
		IF NOT(gT_SafetyStatus.xSetupOperateModeActive) THEN
			(* NormalBetrieb *)
			IF NOT(xMachineDoorUpClose) THEN
				bStateSafetyCtrl:=5;	(* < MaschinenTüre schliessen > *)
			ELSIF NOT(gT_SafetyStatus.xSecuritySwitch) THEN
				bStateSafetyCtrl:=17;	(* < AntriebSperrTaste deaktivieren > *)
			ELSIF NOT(gT_SafetyStatus.xEnergyONNormalMode) AND QxCtrlLampReleaseButton THEN
				bStateSafetyCtrl:=2;	(* < FreigabeTaste drücken > *)
			ELSIF gT_SafetyStatus.xEnergyONNormalMode AND ((dwActualPage = gT_PageNumber.iAutoMode_Process)
			OR (dwActualPage = gT_PageNumber.iAutoMode_ProcessValue1) OR (dwActualPage = gT_PageNumber.iAutoMode_ProcessValue2)		(* IGS *)
			OR (dwActualPage = gT_PageNumber.iAutoMode_PartQuality)) AND TProcess.T_Ctrle.xDone THEN
				IF NOT(gxOnlyCentringActive) AND NOT(gxCentringActive) THEN
					bStateSafetyCtrl:=3;	(* < StartTaste drücken > *)
				ELSIF gxOnlyCentringActive THEN
					bStateSafetyCtrl:=35;	(* < StartTaste drücken (nur Zentrierung Aktiv) > *)
				ELSE
					bStateSafetyCtrl:=36;	(* < StartTaste drücken (Zentrierung + Bearb. Aktiv) > *)
				END_IF;
			ELSIF gT_SafetyStatus.xEnergyONNormalMode AND (dwActualPage = gT_PageNumber.iAutoMode_Referencing) AND TProcess.T_Ctrle.xDone THEN
				bStateSafetyCtrl:=3;	(* < StartTaste drücken > *)
			ELSIF gT_SafetyStatus.xEnergyONNormalMode AND NOT(TProcess.T_Ctrle.xDone) AND (TProcess.T_Ctrle.iFunctNr = 1) THEN
				bStateSafetyCtrl:=26;	(* < Masch.Ref/Grundstellung in Ausführung > *)
			ELSIF gT_SafetyStatus.xEnergyONNormalMode AND NOT(TProcess.T_Ctrle.xDone) AND (TProcess.T_Ctrle.iFunctNr = 2) THEN
				IF NOT(gxOnlyCentringActive) AND NOT(gxCentringActive) THEN
					bStateSafetyCtrl:=25;	(* < Automat in Ausführung > *)
				ELSIF gxOnlyCentringActive THEN
					bStateSafetyCtrl:=37;	(* < Automat in Ausführung (nur Zentrierung Aktiv) > *)
				ELSE
					bStateSafetyCtrl:=38;	(* < Automat in Ausführung (Zentrierung + Bearb. Aktiv) > *)
				END_IF;
			END_IF;
		ELSE
			(* EinrichtBetrieb *)
			IF NOT(gT_SafetyStatus.xSecuritySwitch) THEN
				bStateSafetyCtrl:=17;	(* < AntriebSperrTaste deaktivieren > *)
			ELSIF (gT_SafetyStatus.iSetupMode = 1) AND
			  NOT(gT_SafetyStatus.xEnergyONSetupModeASt1) THEN
				IF gT_SafetyStatus.xSecurityDoorClose THEN
					bStateSafetyCtrl:=2;	(* < FreigabeTaste drücken > *)
				ELSE
					IF T_TwinSafeIn.IxEnablingSwitchActiveCh1 OR T_TwinSafeIn.IxEnablingSwitchActiveCh2 THEN
						xCheckStateEnableSwitch:=TRUE;
					ELSE
						bStateSafetyCtrl:=4;	(* < Zustimmschalter drücken > *)
					END_IF;
				END_IF;
			ELSIF (gT_SafetyStatus.iSetupMode = 2) AND
			  NOT(gT_SafetyStatus.xEnergyONSetupModeBSt1) THEN
				IF gT_SafetyStatus.xSecurityDoorClose THEN
					bStateSafetyCtrl:=2;	(* < FreigabeTaste drücken > *)
				ELSE
					IF T_TwinSafeIn.IxEnablingSwitchActiveCh1 OR T_TwinSafeIn.IxEnablingSwitchActiveCh2 THEN
						xCheckStateEnableSwitch:=TRUE;
					ELSE
						bStateSafetyCtrl:=4;	(* < Zustimmschalter drücken > *)
					END_IF;
				END_IF;
			ELSE
				CASE dwActualPage OF
				gT_PageNumber.iHandMode_Process,gT_PageNumber.iHandMode_WorkParameter,gT_PageNumber.iHandMode_RegulatorPara,gT_PageNumber.iHandMode_OnlineChange,gT_PageNumber.iHandMode_ConfigPosition:
					IF TProcess.T_Ctrle.xDone THEN
						IF NOT(gxOnlyCentringActive) AND NOT(gxCentringActive) THEN
							bStateSafetyCtrl:=3;	(* < StartTaste drücken > *)
						ELSIF gxOnlyCentringActive THEN
							bStateSafetyCtrl:=35;	(* < StartTaste drücken (nur Zentrierung Aktiv) > *)
						ELSE
							bStateSafetyCtrl:=36;	(* < StartTaste drücken (Zentrierung + Bearb. Aktiv) > *)
						END_IF;
					ELSIF NOT(TProcess.T_Ctrle.xDone) AND (TProcess.T_Ctrle.iFunctNr = 3) THEN
						IF NOT(gxOnlyCentringActive) AND NOT(gxCentringActive) THEN
							bStateSafetyCtrl:=28;	(* < HandBetrieb in Ausführung > *)
						ELSIF gxOnlyCentringActive THEN
							bStateSafetyCtrl:=39;	(* < HandBetrieb in Ausführung (nur Zentrierung Aktiv) > *)
						ELSE
							bStateSafetyCtrl:=40;	(* < HandBetrieb in Ausführung (Zentrierung + Bearb. Aktiv) > *)
						END_IF;
					END_IF;
				gT_PageNumber.iHandMode_ProfileMngmt1,gT_PageNumber.iHandMode_ErrorList,gT_PageNumber.iHandMode_Setup1:
					IF NOT(TProcess.T_Ctrle.xDone) AND (TProcess.T_Ctrle.iFunctNr = 3) THEN
						IF NOT(gxOnlyCentringActive) AND NOT(gxCentringActive) THEN
							bStateSafetyCtrl:=28;	(* < HandBetrieb in Ausführung > *)
						ELSIF gxOnlyCentringActive THEN
							bStateSafetyCtrl:=39;	(* < HandBetrieb in Ausführung (nur Zentrierung Aktiv) > *)
						ELSE
							bStateSafetyCtrl:=40;	(* < HandBetrieb in Ausführung (Zentrierung + Bearb. Aktiv) > *)
						END_IF;
					END_IF;
				gT_PageNumber.iWorkStation_Axis1:
					IF TCommonAxis.T_CtrleSingle.xNotMoving THEN
						IF (TCommonAxis.T_Config_Gen.iTyp = 2) OR (TCommonAxis.T_Config_Gen.iTyp = 2) THEN
							IF TCommonAxis.T_CtrleSingle.xPower THEN
								bStateSafetyCtrl:=8;	(* < Für Drehbewegung StartTaste drücken > *)
							ELSE
								bStateSafetyCtrl:=33;	(* < Drehmoment der Achse einschalten > *)
							END_IF;
						ELSE
							IF TCommonAxis.T_CtrleSingle.xRef AND TCommonAxis.T_CtrleSingle.xPower THEN
								bStateSafetyCtrl:=7;	(* < Für Positionsfahrt StartTaste drücken > *)
							ELSIF NOT(TCommonAxis.T_CtrleSingle.xPower) THEN
								bStateSafetyCtrl:=33;	(* < Drehmoment der Achse einschalten > *)
							ELSIF NOT(TCommonAxis.T_CtrleSingle.xRef) THEN
								bStateSafetyCtrl:=34;	(* < Achse Referenzieren für Positionsfahrt > *)
							END_IF;
						END_IF;
					ELSE
						IF (TCommonAxis.T_Config_Gen.iTyp = 2) OR (TCommonAxis.T_Config_Gen.iTyp = 2) THEN
							bStateSafetyCtrl:=9;	(* < Funktion in Ausführung > *)
						ELSE
							bStateSafetyCtrl:=10;	(* < Funktion in Ausführung...MMI ist blockiert > *)
						END_IF;
					END_IF;
				gT_PageNumber.iWorkStation_Cylinder1:
					bStateSafetyCtrl:=22;	(* < Zylinderbewegung EIN/AUS drücken > *)
				gT_PageNumber.iWorkStation_Valve1:
					IF (T_ExchgParam.T_Cylinder.iSelCyl_Setup = 5) THEN
						bStateSafetyCtrl:=20;	(* < Zylinderbewegung mit Joystick bewegen > *)
					ELSE
						bStateSafetyCtrl:=21;	(* < Ventile mit Joystick bewegen > *)
					END_IF;
				gT_PageNumber.iWorkStation_Function1,gT_PageNumber.iWorkStation_Setup1,gT_PageNumber.iWorkStation_Setup2:
					IF xVisuFunctionActive THEN
						bStateSafetyCtrl:=10;	(* < Funktion in Ausführung...MMI ist blockiert > *)
					ELSE
						bStateSafetyCtrl:=3;	(* < StartTaste drücken > *)
					END_IF;
				gT_PageNumber.iWorkStation_Setup3:
					IF xVisuFunctionActive THEN
						bStateSafetyCtrl:=10;	(* < Funktion in Ausführung...MMI ist blockiert > *)
					ELSE
						bStateSafetyCtrl:=3;	(* < StartTaste drücken > *)
					END_IF;
				END_CASE;
			END_IF;
			IF xCheckStateEnableSwitch THEN
				IF (bStateSafetyCtrl = 99) THEN
					TONWaitCheck(IN:=TRUE,PT:=T#100ms);
					IF TONWaitCheck.Q THEN
						bStateSafetyCtrl:=6;	(* < Zustimmtaster lösen > *)
					END_IF;
				END_IF;
			ELSE
				TONWaitCheck(IN:=FALSE);
			END_IF;

		END_IF;
	END_IF;
END_IF;
END_FUNCTION_BLOCK

(* POU GENERAL/FB_CHECKSETUPMODE, ST *)
FUNCTION_BLOCK FB_CHECKSETUPMODE
VAR_INPUT
	T_TwinSafeIn:ST_TWINSAFE_IN;
END_VAR
VAR_OUTPUT
	iSetupMode:INT;	(* 1=A, 2=B, 0=Normalbetrieb *)
END_VAR
VAR
	xSetupModeA: BOOL;
	xSetupModeB: BOOL;
END_VAR
xSetupModeA:=			T_TwinSafeIn.IxKeySwitchProcObservationCh1 AND
						T_TwinSafeIn.IxKeySwitchProcObservationCh2 AND
						NOT(T_TwinSafeIn.IxKeySwitchWorkStationCh1) AND
						NOT(T_TwinSafeIn.IxKeySwitchWorkStationCh2);
xSetupModeB:=			NOT(T_TwinSafeIn.IxKeySwitchProcObservationCh1) AND
						NOT(T_TwinSafeIn.IxKeySwitchProcObservationCh2) AND
						T_TwinSafeIn.IxKeySwitchWorkStationCh1 AND
						T_TwinSafeIn.IxKeySwitchWorkStationCh2;

(* Prozessbeobachtung *)
IF xSetupModeA THEN
	iSetupMode:=1;		(* 1=Prozessbeobachtung *)
(* Bearb.Station *)
ELSIF xSetupModeB THEN
	iSetupMode:=2;		(* 2=Einricht Bearbeitungsstation *)
ELSE
	iSetupMode:=0;		(* 0=Normalbetrieb *)
END_IF;
END_FUNCTION_BLOCK

(* POU GENERAL/FB_CHECKMACHINESTATE, ST *)
FUNCTION_BLOCK FB_CHECKMACHINESTATE
VAR_INPUT
	xSecurityKey:BOOL;		(* state of the keyswitch-->TRUE=EinrichtBetrieb *)
	iSetupMode:INT;			(* Turn switch --> 1=EinrichtBetriebA, 2=EinrichtBetriebB, 0=Normalbetrieb *)
	xNormalOperate_EnergyON:BOOL;
	xSetupOperateA_EnergyON:BOOL;
	xSetupOperateB_EnergyON:BOOL;
END_VAR
VAR_OUTPUT
END_VAR
VAR
	xTmp: BOOL;
END_VAR
T_ExchgParam.T_Visu.bMachineState:=0;
(* Abfragen für Allgemeiner Maschinenzustand *)
xTmp:=	xNormalOperate_EnergyON OR xSetupOperateA_EnergyON OR xSetupOperateB_EnergyON;
xTmp:=	xTmp AND
		TStation_Work_St1.TControl.xReferenced;
IF xTmp THEN
	T_ExchgParam.T_Visu.bMachineState:=T_ExchgParam.T_Visu.bMachineState OR 2#001;		(* 1=Maschine hat keinen Fehler, kein Prozess-/Stationsfunktion aktiv, kein Aktuator ist in Bewegung und die Energieversorgung ist eingeschaltet *)
ELSE
	T_ExchgParam.T_Visu.bMachineState:=T_ExchgParam.T_Visu.bMachineState AND 2#110;
END_IF;
xTmp:=	NOT(TStation_Work_St1.TControl.xDone) OR TStation_Work_St1.TControl.xActiveMovement OR
		T_StartUp.T_State.xBlockChangeMovementVisu OR NOT(T_VisuQVis.T_CtrleProcess.xDone) OR
		NOT(T_VisuQVis.T_CtrleAction.xDone) OR T_VisuQVis.T_CtrleAction.xFunctionActive;
IF xTmp THEN
	T_ExchgParam.T_Visu.bMachineState:=T_ExchgParam.T_Visu.bMachineState OR 2#010;		(* 2=Prozess-/Stationsfunktion Aktiv oder mindestens ein Aktuator ist in Bewegung *)
ELSE
	T_ExchgParam.T_Visu.bMachineState:=T_ExchgParam.T_Visu.bMachineState AND 2#101;
END_IF;
IF (T_ExchgParam.T_Visu.T_Message.iState = 401) THEN
	T_ExchgParam.T_Visu.bMachineState:=T_ExchgParam.T_Visu.bMachineState OR 2#100;		(* 4=Maschine hat mindestens einen Fehler *)
ELSE
	T_ExchgParam.T_Visu.bMachineState:=T_ExchgParam.T_Visu.bMachineState AND 2#011;
END_IF;
END_FUNCTION_BLOCK

(* POU GENERAL/FB_BIOSPARAMETER, ST *)
FUNCTION_BLOCK FB_BIOSPARAMETER
VAR_INPUT
	dwBIOSPasswordPage:DWORD;		(* Page number of the BIOS password page *)
	dwBIOSParameterPage:DWORD;		(* Page number of the BIOS parameter page *)
	xActiveCurrentAxes:BOOL;
	xReadyToSwitchPasswordPage:BOOL;
END_VAR
VAR_IN_OUT
	T_Visu:ST_QVIS;						(* Data structure of the visualisation *)
	T_ExchgParam :ST_QVIS_EXCHG_PARAM;
	T_HDD:ST_HDD;						(* Data structure of the File Management *)
	T_NovRam : ST_NOVRAM;				(* Data structure of the NovRam *)
	T_CtrlePanel:ST_CTRLEPANEL;		(* Data structure of the ControlPanel *)
END_VAR
VAR_OUTPUT
END_VAR
VAR
	TONShowMessage: TON;
	xChangeToBIOSPassword: BOOL;
	xChangeToBIOSParameter: BOOL;
	xSaveBIOSParameterToNovRAM: BOOL;
	xCopyBIOSParameter: BOOL;
	iStepSaveToNovRAM: INT;
	iStepReadFirstTimeParameter: INT;
	xCheckMsgBoxActive: BOOL;
(* Random *)
	fbGetCpuAccount:GETCPUCOUNTER;
	FBPassword_SystemLevel:FB_Password_SystemLevel;
	diPwSystem:DINT;
	xNovRAMParaReaded: BOOL;
END_VAR
(****************************************************************************************************************************************************)
(***********     This Functionblock gives the possibility to set the bios parameter, with input a SystemLevel password     ************)
(****************************************************************************************************************************************************)
xNovRAMParaReaded:=TRUE;
(* Managing BIOS Parameter on Startup *)
	IF (T_ExchgParam.T_Visu.T_Message.iStateBIOS <> 0) THEN
		TONShowMessage(IN:=TRUE,PT:=T#3s);
		IF TONShowMessage.Q THEN
			T_ExchgParam.T_Visu.T_Message.iStateBIOS:=0;
		END_IF;
	ELSE
		TONShowMessage(IN:=FALSE);
	END_IF;
	xCheckMsgBoxActive:=	(T_ExchgParam.T_SafetyCtrl.bStateMessageError <> 0) OR
							(T_ExchgParam.T_SafetyCtrl.bStateMessageInfo <> 0) OR
							(T_ExchgParam.T_SafetyCtrl.bStateMessageWarning <> 0);
	IF ((T_Visu.T_PlcParam.dwActualPage = gT_PageNumber.iStart_Page1) AND NOT(T_Visu.T_CtrleVisu.xExecute) AND T_Visu.T_CtrleVisu.xDone) OR xCheckMsgBoxActive THEN
		xChangeToBIOSPassword:=FALSE;
		xChangeToBIOSParameter:=FALSE;
		xSaveBIOSParameterToNovRAM:=FALSE;
		xCopyBIOSParameter:=FALSE;
		iStepSaveToNovRAM:=1;
		iStepReadFirstTimeParameter:=1;
		T_ExchgParam.T_Visu.T_Message.iStateBIOS:=0;
	END_IF;
	IF (T_Visu.T_PlcParam.dwActualPage = dwBIOSPasswordPage) OR (T_Visu.T_PlcParam.dwActualPage = dwBIOSParameterPage) THEN
		IF xActiveCurrentAxes THEN	(* check if external relase button has been pressed *)
			IF NOT(T_Visu.T_CtrleVisu.xExecute) AND T_Visu.T_CtrleVisu.xDone THEN
				T_Visu.T_PlcParam.dwSetNewPage:=0;
				T_Visu.T_CtrleVisu.iFunction:=1;
				T_Visu.T_CtrleVisu.xExecute:=TRUE;
			END_IF;
		END_IF;
	END_IF;
	(* check if the function button is pressed-->if it is pressed the change to the BIOS password page *)
	IF NOT(xChangeToBIOSPassword) THEN
		IF (T_Visu.T_PlcParam.dwActualPage = gT_PageNumber.iStart_Page1) AND NOT(T_StartUp.T_State.xCompleted) AND NOT(xCheckMsgBoxActive) THEN
			IF T_ExchgParam.T_BtFunctionPanel.wActivBt = 16#1 THEN
				T_ExchgParam.T_BtFunctionPanel.wActivBt:=0;
				IF NOT(xActiveCurrentAxes) THEN
					IF NOT(gxAxisPositionSettled) THEN
						IF NOT(T_Visu.T_CtrleVisu.xExecute) AND T_Visu.T_CtrleVisu.xDone THEN
							T_ExchgParam.T_Visu.T_Message.iStateBIOS:=0;
							xChangeToBIOSPassword:=TRUE;
							T_Visu.T_PlcParam.dwSetNewPage:=dwBIOSPasswordPage;
							T_Visu.T_CtrleVisu.iFunction:=1;
							T_Visu.T_CtrleVisu.xExecute:=TRUE;
							(* Der Counter respektive Random muss 9 Stellig sein welches aus dem Zyklusticker der CPU ausgelesen wird *)
							fbGetCpuAccount;
							FBPassword_SystemLevel(	dwCounterHI:= fbGetCpuAccount.cpuCntHiDW,
													dwCounterLOW:=fbGetCpuAccount.cpuCntLoDW);
							T_ExchgParam.T_Visu.T_Level.diRandom:=FBPassword_SystemLevel.diRandom;
							diPwSystem:=FBPassword_SystemLevel.diPwSystem;
						END_IF;
					ELSE
						T_ExchgParam.T_Visu.T_Message.iState:=225;	(* Warnung: BIOS Parameter nur vor dem erstmaligen Booten zugänglich ! *)
					END_IF;
				ELSE
					T_ExchgParam.T_Visu.T_Message.iState:=226;	(* Warnung: BIOS Parameter nur bei ausgeschalteter Energieversorgung ! *)
				END_IF;
			END_IF;
		END_IF;
	END_IF;
	(* check the settled password *)
	IF xChangeToBIOSPassword THEN
		IF (T_Visu.T_PlcParam.dwActualPage = dwBIOSPasswordPage) THEN
			IF T_ExchgParam.T_Visu.xKey_Escape THEN	(* ESC Button for exit and go to the Startpage *)
				T_ExchgParam.T_Visu.xKey_Escape:=FALSE;
				IF NOT(T_Visu.T_CtrleVisu.xExecute) AND T_Visu.T_CtrleVisu.xDone THEN
					xChangeToBIOSPassword:=FALSE;
					T_Visu.T_PlcParam.dwSetNewPage:=0;
					T_Visu.T_CtrleVisu.iFunction:=1;
					T_Visu.T_CtrleVisu.xExecute:=TRUE;
					T_ExchgParam.T_Visu.T_Level.diPwSystem:=-1;
				END_IF;
			END_IF;
			IF (T_ExchgParam.T_Visu.T_Level.diPwSystem = diPwSystem) THEN
				T_ExchgParam.T_Visu.T_Message.iStateBIOS:=0;
				T_ExchgParam.T_Visu.T_Level.diPwSystem:=-1;
				IF NOT(T_Visu.T_CtrleVisu.xExecute) AND T_Visu.T_CtrleVisu.xDone THEN
					xChangeToBIOSPassword:=FALSE;
					xChangeToBIOSParameter:=TRUE;
					T_Visu.T_PlcParam.dwSetNewPage:=dwBIOSParameterPage;
					T_Visu.T_CtrleVisu.iFunction:=1;
					T_Visu.T_CtrleVisu.xExecute:=TRUE;
					xCopyBIOSParameter:=TRUE;
					T_CtrlePanel.udiButton:=0;
				END_IF;
			END_IF;
			IF (T_ExchgParam.T_Visu.T_Level.diPwSystem <> -1) THEN
				IF (T_ExchgParam.T_Visu.T_Level.diPwSystem <> diPwSystem) THEN
					T_ExchgParam.T_Visu.T_Message.iStateBIOS:=2;	(* Falsches Passwort *)
					T_ExchgParam.T_Visu.T_Level.diPwSystem:=-1;
					(* Der Counter respektive Random muss 9 Stellig sein welches aus dem Zyklusticker der CPU ausgelesen wird *)
					fbGetCpuAccount;
					FBPassword_SystemLevel(	dwCounterHI:= fbGetCpuAccount.cpuCntHiDW,
											dwCounterLOW:=fbGetCpuAccount.cpuCntLoDW);
					T_ExchgParam.T_Visu.T_Level.diRandom:=FBPassword_SystemLevel.diRandom;
					diPwSystem:=FBPassword_SystemLevel.diPwSystem;
				END_IF;
			END_IF;
		END_IF;
	END_IF;
	(* the edit parameterlist is now active *)
	IF xChangeToBIOSParameter THEN
		IF (T_Visu.T_PlcParam.dwActualPage = dwBIOSParameterPage) AND NOT(xSaveBIOSParameterToNovRAM) AND NOT(xCopyBIOSParameter) THEN
			IF T_ExchgParam.T_Visu.xKey_Escape THEN	(* ESC Button for exit and go to the Startpage *)
				T_ExchgParam.T_Visu.xKey_Escape:=FALSE;
				IF NOT(T_Visu.T_CtrleVisu.xExecute) AND T_Visu.T_CtrleVisu.xDone THEN
					xChangeToBIOSParameter:=FALSE;
					xSaveBIOSParameterToNovRAM:=FALSE;
					xCopyBIOSParameter:=TRUE;
					T_Visu.T_PlcParam.dwSetNewPage:=0;
					T_Visu.T_CtrleVisu.iFunction:=1;
					T_Visu.T_CtrleVisu.xExecute:=TRUE;
				END_IF;
			END_IF;
			IF (UDINT_TO_WORD(T_CtrlePanel.udiButton) = 16#200) AND NOT(xSaveBIOSParameterToNovRAM) THEN	(* Right Panel Button for save Parameter *)
				T_CtrlePanel.udiButton:=0;
				T_ExchgParam.T_Visu.T_Message.iStateBIOS:=1;	(* Parameter gespeichert *)
				xSaveBIOSParameterToNovRAM:=TRUE;
				xCopyBIOSParameter:=FALSE;
				iStepSaveToNovRAM:=1;
			END_IF;
		END_IF;
	END_IF;
	(* save the settled parameter to the NovRam *)
	IF xSaveBIOSParameterToNovRAM THEN
		CASE iStepSaveToNovRAM OF
		1:	IF xNovRAMParaReaded THEN
				T_NovRam.T_Parameter.T_StationWork[gciStationSt1].T_AxisState.xReferencedZAxis:=T_ExchgParam.T_ParamBIOS.xReferencedZAxis_St1;
				T_NovRAM.T_Ctrle.iFunction:=2;
				T_NovRAM.T_Ctrle.xExecute:=TRUE;
				iStepSaveToNovRAM:=10;
			ELSE
				iStepSaveToNovRAM:=1;
				xSaveBIOSParameterToNovRAM:=FALSE;
			END_IF;
		10:	IF NOT(T_NovRAM.T_Ctrle.xExecute) AND T_NovRAM.T_Ctrle.xDone THEN
				iStepSaveToNovRAM:=1;
				xSaveBIOSParameterToNovRAM:=FALSE;
				T_Visu.T_CtrleVisu.xReset:=TRUE;	(* Exit the BIOS Parameter Page *)
			END_IF;
		END_CASE;
	END_IF;
	(* copy the NovRam config parameter to the visu structure *)
	IF xCopyBIOSParameter THEN
		IF xNovRAMParaReaded THEN
			T_ExchgParam.T_ParamBIOS.xReferencedZAxis_St1:=T_NovRam.T_Parameter.T_StationWork[gciStationSt1].T_AxisState.xReferencedZAxis;
			xCopyBIOSParameter:=FALSE;
		ELSE
			xCopyBIOSParameter:=FALSE;
		END_IF;
	END_IF;
END_FUNCTION_BLOCK

(* POU GENERAL/FB_Password_SystemLevel, ST *)
FUNCTION_BLOCK FB_Password_SystemLevel
VAR_INPUT
	dwCounterHI:DWORD;
	dwCounterLOW:DWORD;
END_VAR
VAR_OUTPUT
	diRandom:DINT;
	diPwSystem:DINT;
END_VAR
VAR
	ii:INT;
	diCounter:DINT;
	sTmp:STRING;
	sValueHighAndLow: STRING;
	iMissingPlace: INT;
END_VAR
(*
	dynamic System password
	ex : Counter=123456789 => pw=825
	formul : 1+2+3+4+5+6+7+8+9+ 80 + 700 = 825
*)

(* Init. value *)
	diPwSystem:=0;
(* Convert value *)
	(* Counter auf 9 Stellig definieren *)
	IF (dwCounterHI <> 0) AND (dwCounterLOW <> 0) THEN
		sValueHighAndLow:=CONCAT(DWORD_TO_STRING(dwCounterHI),DWORD_TO_STRING(dwCounterLOW));
	ELSIF (dwCounterHI = 0) AND (dwCounterLOW <> 0) THEN
		sValueHighAndLow:=DWORD_TO_STRING(dwCounterLOW);
	ELSIF (dwCounterHI <> 0) AND (dwCounterLOW = 0) THEN
		sValueHighAndLow:=DWORD_TO_STRING(dwCounterHI);
	ELSE
		sValueHighAndLow:='';
	END_IF;
	IF (LEN(sValueHighAndLow) >= 9) THEN
		diCounter:=STRING_TO_DINT(MID(sValueHighAndLow,9,LEN(sValueHighAndLow)-8));
	ELSE
		(* Fehlende Zeichen noch aufüllen bis 9 Zeichen *)
		iMissingPlace:=LEN(sValueHighAndLow);
		FOR ii:=1 TO 9 - iMissingPlace DO
			sValueHighAndLow:=CONCAT(INT_TO_STRING(ii),sValueHighAndLow);
		END_FOR;
		diCounter:=STRING_TO_DINT(sValueHighAndLow);
	END_IF;

(* Set Random value *)
	diRandom:=diCounter;
	sTmp:=DINT_TO_STRING(diCounter);
(* Set System pw *)
	FOR ii:=0 TO LEN(sTmp)-1 DO
		diPwSystem:=diPwSystem+STRING_TO_DINT(MID(sTmp,1,LEN(sTmp)-ii));
		IF ii=1 THEN diPwSystem:=diPwSystem+STRING_TO_DINT(MID(sTmp,1,LEN(sTmp)-ii))*10; END_IF
		IF ii=2 THEN diPwSystem:=diPwSystem+STRING_TO_DINT(MID(sTmp,1,LEN(sTmp)-ii))*100; END_IF
	END_FOR
END_FUNCTION_BLOCK

(* POU PRG_LAYER2_HARDWARE/FBHWSTATIONEN/FBHW_STATION_WORK, ST *)
FUNCTION_BLOCK FBHW_STATION_WORK
VAR_INPUT
	iStationNr:INT;
	(* IO's *)
	xStationPowerON:BOOL;
	IxToolDeflection:BOOL;	(* Überwachung der Werkzeug Auslenkung für die Werkzeug Spindel *)
	IiAToolTorque:INT;	(* Drehmoment Sensor für Drehmomentüberwachung für die Werkzeug Spindel *)
	IiAToolTorque2:INT;	(* Drehmoment Sensor für Drehmomentüberwachung für die Werkzeug Spindel *)	(* IGS *)
	IxBrakeReleaseZAxis:BOOL;	(* Sensor für Bremse gelöst bei der Z Achse (Hubachse) *)
	IxUpperToolGuide_WorkpieceClamped:BOOL;	(* Sensor für Überwachung der Werkstückfixierung *)
	IbTooSpindleActive:BYTE;																		(* IGS *)
	iSlaveAddr_AxisZ:INT;
	iSlaveAddr_AxisS:INT;																			(* IGS *)
	IxTorqueOverload:BOOL;			(* Clock-->Signal induktiver Sensor für Drehmomentüberlast *)			(* IGS *)
END_VAR
VAR_IN_OUT
	T_Station_Parameter: ST_RETAIN_DATA_STATIONWORK;
	T_Station_Work : ST_STATION;
	(* Axis value *)
	IuiActualTorqueAxisZ :UINT;
	IwInputState_Z_Axis:WORD;
	IuiActualTorqueAxisS :UINT;
	IwInputState_S1_Axis:WORD;
	IwInputState_S2_Axis:WORD;									(* IGS *)
	IwInputState_S3_Axis:WORD;									(* IGS *)
	(* Axis structure *)
	stZRefIn :NCTOPLC_AXLESTRUCT;
	stZRefOut :PLCTONC_AXLESTRUCT;
	stZDriveState :ST_AXIS_DRIVESTATE;
	stSRefIn :NCTOPLC_AXLESTRUCT;
	stSRefOut :PLCTONC_AXLESTRUCT;
	stS2RefIn :NCTOPLC_AXLESTRUCT;	(* Beckhoff Spindel *)		(* IGS *)
	stS2RefOut :PLCTONC_AXLESTRUCT;	(* Beckhoff Spindel *)		(* IGS *)
	stS3RefIn :NCTOPLC_AXLESTRUCT;	(* Beckhoff Spindel *)		(* IGS *)
	stS3RefOut :PLCTONC_AXLESTRUCT;	(* Beckhoff Spindel *)		(* IGS *)
	T_HDD : ST_HDD;
	T_TwinSafe_Ctrle_Z_Axis:ST_TWINSAFE_DRIVE;
	T_TwinSafe_Status_Z_Axis:ST_TWINSAFE_DRIVE;
	T_TwinSafe_Ctrle_S2_Axis:ST_TWINSAFE_DRIVE;				(* IGS *)
	T_TwinSafe_Status_S2_Axis:ST_TWINSAFE_DRIVE;				(* IGS *)
	T_TwinSafe_Ctrle_S3_Axis:ST_TWINSAFE_DRIVE;				(* IGS *)
	T_TwinSafe_Status_S3_Axis:ST_TWINSAFE_DRIVE;				(* IGS *)
	(* Axis DC structure *)
	stBubblerDataIN : ST_COMM_IN_DCAXIS;						(* IGS3 *)
	stBubblerDataOUT : ST_COMM_OUT_DCAXIS;					(* IGS3 *)
	stFeedpumpINData : ST_COMM_IN_DCAXIS;						(* IGS3 *)
	stFeedpumpOUTData : ST_COMM_OUT_DCAXIS;					(* IGS3 *)
END_VAR
VAR_OUTPUT
	xActiveHWStation : BOOL;
	xActiveStation : BOOL;
	xEnableMasterModul:BOOL;	(* is for the Shuttle Axis *)
	QiAToolDeflection_SM:INT;
	QiAToolTorqueHC_SM:INT;
	QiAToolTorqueOverload_SM:INT;
	QxCylBrakeReleaseZAxis_Open:BOOL;	(* Ventil für Bremszylinder der Z(St1) Achse für Bremse lösen *)
	QxCylBrakeReleaseZAxis_Close:BOOL;	(* Ventil für Bremszylinder der Z(St1) Achse für Bremse aktivieren *)
	QxCylWorkpieceClamp_Open:BOOL;	(* Ventil für Werkstückfixierzylinder öffnen *)
	QxCylWorkpieceClamp_Close:BOOL;	(* Ventil für Werkstückfixierzylinder schliessen *)
	QxAirTable:BOOL;	(* Ventil für die Luft des Tisches *)
	QxVacuumTable:BOOL;	(* Ventil für das Vakuum des Tisches *)
	QxMeasRangeTorqueSensor:BOOL;		(* Drehmoment Sensor Bereichsumschaltung von 0-2Nm auf 0-0.5Nm *)		(* IGS *)
	QxControlTorqueSensor:BOOL;			(* Drehmoment Sensor Kontrollfunktion aktivieren *)						(* IGS *)
END_VAR
VAR
(* Pointer auf Actuatoren *)
	ptrTAxisZ 							:POINTER TO ST_AXIS;			(* Achse für die Hubachse *)
	ptrTAxisS 							:POINTER TO ST_AXIS;			(* Achse für die Werkzeugspindel *)
	ptrTCylToolDeflection					:POINTER TO ST_CYLINDER;	(* Servoventil für das bestimmen der vertikalen Auslenkraft *)
	ptrTCylToolTorqueHC 					:POINTER TO ST_CYLINDER;	(* Drehmomentueberwachung HC *)
	ptrTCylToolTorqueOverload 			:POINTER TO ST_CYLINDER;	(* Drehmomentueberwachung Ueberlast *)
	ptrTTorqueSensorMeasRange			:POINTER TO ST_CYLINDER;	(* Controlling für den Drehmomentsensor, Einstellung des Drehmomentbereiches *)	(* IGS *)
	ptrTTorqueSensorControl				:POINTER TO ST_CYLINDER;	(* Controlling für den Drehmomentsensor, Ueberpruefung auf Funktionalitaet *)			(* IGS *)
	ptrTSensorTorque 					:POINTER TO ST_CYLINDER;	(* Analoger Sensor für Drehmoment detektion *)
	ptrTSensorTorqueOverload 			:POINTER TO ST_CYLINDER;	(* Digitaler Sensor für Drehmoment Ueberlast detektion *)							(* IGS *)
	ptrTCylBrakeReleaseZAxis 				:POINTER TO ST_CYLINDER;	(* Zylinder für lösen der Bremse bei der Z Achse *)
	ptrTCylWorkpieceClamp				:POINTER TO ST_CYLINDER;	(* Ventil fuer Werkstueckfixierzylinder *)
	ptrTValveAirTable						:POINTER TO ST_CYLINDER;	(* Ventil fuer die Luft des Tisches *)
	ptrTValveVacuumTable				:POINTER TO ST_CYLINDER;	(* Ventil fuer die Luft des Tisches *)
	ptrTValveCleanNozzle					:POINTER TO ST_CYLINDER;	(* Ventil fuer die Reinigungsduese *)											(* BEF *)
	ptrTAxisBubbler						:POINTER TO ST_DC_AXIS;	(* Ruehrwerk fuer Suspension *)												(* IGS3 *)
	ptrTAxisFeedPump					:POINTER TO ST_DC_AXIS;	(* Foerderpumpe fuer Suspension *)											(* IGS3 *)

(* Functionblock axis *)
	fbAxisZ:FBHW_AXIS_SINGLE;
	fbAxisZLiveValues:FBHW_AXIS_LIVEVALUES;
	fbAxisToolSpindleS: FBHW_AXIS_SINGLE;
	fbAxisToolSpindleSLiveValues: FBHW_AXIS_LIVEVALUES;
	(* DC Motor Maxon *)
	fbBubbler:FBHW_AXIS_DC;			(* Motor für das Rührwerk der Suspension *)		(* IGS3 *)
	fbFeedpump:FBHW_AXIS_DC;		(* Motor für die Förderpumpe der Suspension *)		(* IGS3 *)
(* Functionblock cylinder *)
	fbCylToolDeflection : FBHW_CYL_ANALOG;
	fbCylToolTorqueHC : FBHW_CYL_ANALOG;
	fbCylToolTorqueOverload : FBHW_CYL_ANALOG;
	fbTorqueSensorMeasRange	:FBHW_CYL_STANDARD;		(* IGS *)
	fbTorqueSensorControl		:FBHW_CYL_STANDARD;		(* IGS *)
	FBCalcSpindleForce: FB_CalcSpindleForce;
	FBTorqueLevelAirPressureAnalog_HC:FB_TorqueLevelAirPressureAnalog;
	FBTorqueLevelAirPressureAnalog_Overload:FB_TorqueLevelAirPressureAnalog;
	fbCylTBrakeReleaseZAxis : FBHW_CYL_STANDARD_2WAY;
	fbCylWorkpieceClamp : FBHW_CYL_STANDARD_2WAY;
	fbValveAirTable : FBHW_CYL_STANDARD;
	fbValveVacuumTable : FBHW_CYL_STANDARD;
	fbValveCleanNozzle : FBHW_CYL_STANDARD;
	iStepResetHardware: INT;
	xHardwareActive: BOOL;
	TONWaitTimeOut: TON;
	RisingEdgeHWConfig: R_TRIG;
	xHardwareConfigError: BOOL;
	xCkeckAcitveMovement: BOOL;
	TONTickTime: TON;
	iStepCountError: INT;
	FBReadAxisState: FB_ReadAxisState;
	rCalcForceIn: REAL;
	T_RegulatorSpindle:ST_EXCHG_PARAM_CONTRMOT;
	FBWriteObject: FB_WriteObject;
	ii:INT;
	rDefaultValue: REAL;
	rQualitySum: REAL;
	rQualityArea: REAL;
	jj: INT;
	rQuality: REAL;
	TONWaitCycle: TON;
	xFirstTime: BOOL;
	TONCalcImpuls: TON;
	xInitCountHC: BOOL;
	xTorqueActive: BOOL;
	xSetParameter: BOOL;
	xInitState: BOOL;															(* IGS *)
	udiTorqueOverloadCounterValue:UDINT;										(* IGS *)
	TOFSetOutput:TOF;														(* IGS *)
	(* .A01_AX5000_Parametrization *)
	fbGetAmsNetID				:FB_GetAxisAmsAddr;							(* IGS *)
	fbSetSlaveState				:FB_EcSetSlaveState;							(* IGS *)
	fbGetSlaveState				:FB_EcGetSlaveState;							(* IGS *)
	fbSoERead					:FB_EcSoERead;								(* IGS *)
	fbSoEWrite					:FB_EcSoEWrite;								(* IGS *)
	sEtherCATNetId 				:STRING;	(*Master Ethercat AMS Adress *)		(* IGS *)
	xReadSoEParameter:BOOL;												(* IGS *)
	iStepReadSoEParameter:INT;												(* IGS *)
	iStepWriteSoEParameter:INT;												(* IGS *)
	lrCalcSpeed: LREAL;
	lrActualSpeed: LREAL;
	lrCheckSpeed: LREAL;
	lrCtrlSpeed: LREAL;
	xZMovementNOK: BOOL;
	TONCheckMovement: TON;
	diCounterTest: DINT;
END_VAR
(****************************************************************************************************************************************************)
(***********                                            This Functionblock manage all the machine hardware                                                           ************)
(****************************************************************************************************************************************************)
T_Station_Work.iStationNr:=iStationNr;
IF T_Station_Work.TControl.xResetHardware THEN
	CASE iStepResetHardware OF
		1:	iStepCountError:=iStepCountError + 1;
			xHardwareActive:=T_Station_Work.TControl.xActiveHardware;
			T_Station_Work.TControl.xActiveHardware:=TRUE;
			iStepResetHardware:=iStepResetHardware + 1;
		2:	T_Station_Work.THWWorkStation.TAxisZ.T_CtrleSingle.xReset:=TRUE;
			T_Station_Work.THWWorkStation.TAxisS.T_CtrleSingle.xReset:=TRUE;
			IF NOT(xSetParameter) AND (T_ExchgParam.bToolSpindleActive = 1) THEN		(* nur laden wenn Maxon Spindel aktiv ist *)
				iStepResetHardware:=iStepResetHardware + 1;
			ELSE
				iStepResetHardware:=iStepResetHardware + 2;
			END_IF;
		3:	T_RegulatorSpindle:=T_Station_Parameter.T_RegulatorSpindle_SM;
			FBWriteObject(	bExecute:= TRUE,
							iFunctionNr:= 1,
							nSlaveAddr:= iSlaveAddr_AxisS,
							T_RegulatorSpindle:= T_RegulatorSpindle,
							T_AxisRefIn:= stSRefIn);
			IF FBWriteObject.Done THEN
				iStepResetHardware:=iStepResetHardware + 1;
				FBWriteObject(	bExecute:=FALSE,
								T_AxisRefIn:= stSRefIn);
				xSetParameter:=TRUE;
			END_IF;


		4:	FBReadAxisState(	bExecute:= TRUE,
								iFunctionNr:= 1,
								nSlaveAddr:=iSlaveAddr_AxisZ,
								nSubIndex:=7,		(* Stauts für Z Achse *)
								T_AxisRefIn:= stZRefIn);
			IF FBReadAxisState.Done THEN
				iStepResetHardware:=iStepResetHardware + 1;
				FBReadAxisState(	bExecute:=FALSE,
								T_AxisRefIn:= stZRefIn);
				IF ((FBReadAxisState.dwValueOut AND 16#FF00) = 16#9000) THEN
					T_ExchgParam.T_Visu.T_Message.iState:=310;	(* Warnung: Z Achse: SLS Sicherheitsfunktion aktiviert ! *)
				END_IF;
			END_IF;
		5:	IF (T_ExchgParam.bToolSpindleActive <> 1) THEN	(* nur ausführen wenn nicht Maxon Spindel aktiv ist *)
				CASE T_ExchgParam.bToolSpindleActive OF
				2:	FBReadAxisState(	bExecute:= TRUE,
									iFunctionNr:= 1,
									nSlaveAddr:=iSlaveAddr_AxisS,
									nSubIndex:=7,		(* Stauts für S2 Achse *)
									T_AxisRefIn:= stS2RefIn);
				3:	FBReadAxisState(	bExecute:= TRUE,
									iFunctionNr:= 1,
									nSlaveAddr:=iSlaveAddr_AxisS,
									nSubIndex:=8,		(* Stauts für S3 Achse *)
									T_AxisRefIn:= stS3RefIn);
				END_CASE;
			END_IF;
			IF FBReadAxisState.Done THEN
				iStepResetHardware:=iStepResetHardware + 1;
				CASE T_ExchgParam.bToolSpindleActive OF
				2:	FBReadAxisState(	bExecute:=FALSE,
									T_AxisRefIn:= stS2RefIn);
				3:	FBReadAxisState(	bExecute:=FALSE,
									T_AxisRefIn:= stS3RefIn);
				END_CASE;
				IF ((FBReadAxisState.dwValueOut AND 16#FF00) = 16#9000) THEN
					T_ExchgParam.T_Visu.T_Message.iState:=311;	(* Warnung: S Achse: SLS Sicherheitsfunktion aktiviert ! *)
				END_IF;
			END_IF;

